Fanuc TP program (LS listing): CODE5.ls

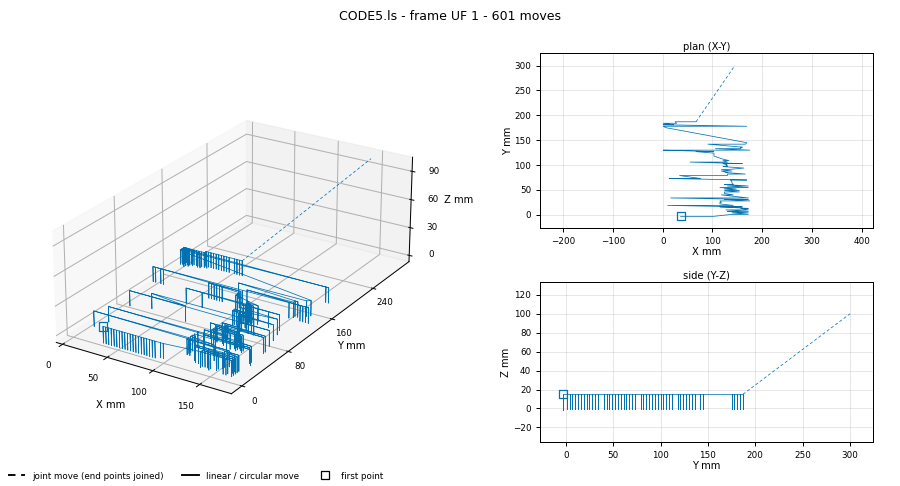
[picture p0: tool path of CODE5.ls in frame UF 1, 601 of 601 moves have a stored position in this frame; points joined in program order, loops and branches not executed]
/PROG CODE5
/ATTR
OWNER		= NOC_FANU;
COMMENT		= "NOC_FANUC";
PROG_SIZE	= 328;
CREATE		= DATE 97-07-08  TIME 03:05:20;
MODIFIED	= DATE 17-07-08  TIME 03:05:26;
FILE_NAME	= ;
VERSION		= 0;
LINE_COUNT	= 10;
MEMORY_SIZE	= 692;
PROTECT		= READ_WRITE;
TCD:  STACK_SIZE	= 0,
      TASK_PRIORITY	= 0,
      TIME_SLICE	= 0,
      BUSY_LAMP_OFF	= 0,
      ABORT_REQUEST	= 0,
      PAUSE_REQUEST	= 0;
DEFAULT_GROUP	= 1,*,*,*,*;
CONTROL_CODE	= 00000000 00000000;
/APPL
/MN
1:UFRAME_NUM=1 ;
2:UTOOL_NUM=5;
3:J P[265] 10% CNT100;
4:L P[266] 250mm/sec FINE;
5:L P[267] 250mm/sec CNT100;
6:L P[268] 250mm/sec CNT100;
7:L P[269] 250mm/sec FINE;
8:L P[270] 250mm/sec CNT100;
9:L P[271] 250mm/sec CNT100;
10:L P[272] 250mm/sec FINE;
11:L P[273] 250mm/sec CNT100;
12:L P[274] 250mm/sec CNT100;
13:L P[275] 250mm/sec FINE;
14:L P[276] 250mm/sec CNT100;
15:L P[277] 250mm/sec CNT100;
16:L P[278] 250mm/sec FINE;
17:L P[279] 250mm/sec CNT100;
18:L P[280] 250mm/sec CNT100;
19:L P[281] 250mm/sec FINE;
20:L P[282] 250mm/sec CNT100;
21:L P[283] 250mm/sec CNT100;
22:L P[284] 250mm/sec FINE;
23:L P[285] 250mm/sec CNT100;
24:L P[286] 250mm/sec CNT100;
25:L P[287] 250mm/sec FINE;
26:L P[288] 250mm/sec CNT100;
27:L P[289] 250mm/sec CNT100;
28:L P[290] 250mm/sec FINE;
29:L P[291] 250mm/sec CNT100;
30:L P[292] 250mm/sec CNT100;
31:L P[293] 250mm/sec FINE;
32:L P[294] 250mm/sec CNT100;
33:L P[295] 250mm/sec CNT100;
34:L P[296] 250mm/sec FINE;
35:L P[297] 250mm/sec CNT100;
36:L P[298] 250mm/sec CNT100;
37:L P[299] 250mm/sec FINE;
38:L P[300] 250mm/sec CNT100;
39:L P[301] 250mm/sec CNT100;
40:L P[302] 250mm/sec FINE;
41:L P[303] 250mm/sec CNT100;
42:L P[304] 250mm/sec CNT100;
43:L P[305] 250mm/sec FINE;
44:L P[306] 250mm/sec CNT100;
45:L P[307] 250mm/sec CNT100;
46:L P[308] 250mm/sec FINE;
47:L P[309] 250mm/sec CNT100;
48:L P[310] 250mm/sec CNT100;
49:L P[311] 250mm/sec FINE;
50:L P[312] 250mm/sec CNT100;
51:L P[313] 250mm/sec CNT100;
52:L P[314] 250mm/sec FINE;
53:L P[315] 250mm/sec CNT100;
54:L P[316] 250mm/sec CNT100;
55:L P[317] 250mm/sec FINE;
56:L P[318] 250mm/sec CNT100;
57:L P[319] 250mm/sec CNT100;
58:L P[320] 250mm/sec FINE;
59:L P[321] 250mm/sec CNT100;
60:L P[322] 250mm/sec CNT100;
61:L P[323] 250mm/sec FINE;
62:L P[324] 250mm/sec CNT100;
63:L P[325] 250mm/sec CNT100;
64:L P[326] 250mm/sec FINE;
65:L P[327] 250mm/sec CNT100;
66:L P[328] 250mm/sec CNT100;
67:L P[329] 250mm/sec FINE;
68:L P[330] 250mm/sec CNT100;
69:L P[535] 250mm/sec CNT100;
70:L P[536] 250mm/sec FINE;
71:L P[537] 250mm/sec CNT100;
72:L P[538] 250mm/sec CNT100;
73:L P[539] 250mm/sec FINE;
74:L P[540] 250mm/sec CNT100;
75:L P[541] 250mm/sec CNT100;
76:L P[542] 250mm/sec FINE;
77:L P[543] 250mm/sec CNT100;
78:L P[544] 250mm/sec CNT100;
79:L P[545] 250mm/sec FINE;
80:L P[546] 250mm/sec CNT100;
81:L P[550] 250mm/sec CNT100;
82:L P[551] 250mm/sec FINE;
83:L P[552] 250mm/sec CNT100;
84:L P[697] 250mm/sec CNT100;
85:L P[698] 250mm/sec FINE;
86:L P[699] 250mm/sec CNT100;
87:L P[700] 250mm/sec CNT100;
88:L P[701] 250mm/sec FINE;
89:L P[702] 250mm/sec CNT100;
90:L P[703] 250mm/sec CNT100;
91:L P[704] 250mm/sec FINE;
92:L P[705] 250mm/sec CNT100;
93:L P[706] 250mm/sec CNT100;
94:L P[707] 250mm/sec FINE;
95:L P[708] 250mm/sec CNT100;
96:L P[712] 250mm/sec CNT100;
97:L P[713] 250mm/sec FINE;
98:L P[714] 250mm/sec CNT100;
99:L P[715] 250mm/sec CNT100;
100:L P[716] 250mm/sec FINE;
101:L P[717] 250mm/sec CNT100;
102:L P[718] 250mm/sec CNT100;
103:L P[719] 250mm/sec FINE;
104:L P[720] 250mm/sec CNT100;
105:L P[856] 250mm/sec CNT100;
106:L P[857] 250mm/sec FINE;
107:L P[858] 250mm/sec CNT100;
108:L P[859] 250mm/sec CNT100;
109:L P[860] 250mm/sec FINE;
110:L P[861] 250mm/sec CNT100;
111:L P[868] 250mm/sec CNT100;
112:L P[869] 250mm/sec FINE;
113:L P[870] 250mm/sec CNT100;
114:L P[874] 250mm/sec CNT100;
115:L P[875] 250mm/sec FINE;
116:L P[876] 250mm/sec CNT100;
117:L P[877] 250mm/sec CNT100;
118:L P[878] 250mm/sec FINE;
119:L P[879] 250mm/sec CNT100;
120:L P[1012] 250mm/sec CNT100;
121:L P[1013] 250mm/sec FINE;
122:L P[1014] 250mm/sec CNT100;
123:L P[1027] 250mm/sec CNT100;
124:L P[1028] 250mm/sec FINE;
125:L P[1029] 250mm/sec CNT100;
126:L P[1033] 250mm/sec CNT100;
127:L P[1034] 250mm/sec FINE;
128:L P[1035] 250mm/sec CNT100;
129:L P[1036] 250mm/sec CNT100;
130:L P[1037] 250mm/sec FINE;
131:L P[1038] 250mm/sec CNT100;
132:L P[1039] 250mm/sec CNT100;
133:L P[1040] 250mm/sec FINE;
134:L P[1041] 250mm/sec CNT100;
135:L P[1192] 250mm/sec CNT100;
136:L P[1193] 250mm/sec FINE;
137:L P[1194] 250mm/sec CNT100;
138:L P[1195] 250mm/sec CNT100;
139:L P[1196] 250mm/sec FINE;
140:L P[1197] 250mm/sec CNT100;
141:L P[1198] 250mm/sec CNT100;
142:L P[1199] 250mm/sec FINE;
143:L P[1200] 250mm/sec CNT100;
144:L P[1318] 250mm/sec CNT100;
145:L P[1319] 250mm/sec FINE;
146:L P[1320] 250mm/sec CNT100;
147:L P[1321] 250mm/sec CNT100;
148:L P[1322] 250mm/sec FINE;
149:L P[1323] 250mm/sec CNT100;
150:L P[1348] 250mm/sec CNT100;
151:L P[1349] 250mm/sec FINE;
152:L P[1350] 250mm/sec CNT100;
153:L P[1369] 250mm/sec CNT100;
154:L P[1370] 250mm/sec FINE;
155:L P[1371] 250mm/sec CNT100;
156:L P[1474] 250mm/sec CNT100;
157:L P[1475] 250mm/sec FINE;
158:L P[1476] 250mm/sec CNT100;
159:L P[1501] 250mm/sec CNT100;
160:L P[1502] 250mm/sec FINE;
161:L P[1503] 250mm/sec CNT100;
162:L P[1624] 250mm/sec CNT100;
163:L P[1625] 250mm/sec FINE;
164:L P[1626] 250mm/sec CNT100;
165:L P[1771] 250mm/sec CNT100;
166:L P[1772] 250mm/sec FINE;
167:L P[1773] 250mm/sec CNT100;
168:L P[1774] 250mm/sec CNT100;
169:L P[1775] 250mm/sec FINE;
170:L P[1776] 250mm/sec CNT100;
171:L P[1915] 250mm/sec CNT100;
172:L P[1916] 250mm/sec FINE;
173:L P[1917] 250mm/sec CNT100;
174:L P[1945] 250mm/sec CNT100;
175:L P[1946] 250mm/sec FINE;
176:L P[1947] 250mm/sec CNT100;
177:L P[2071] 250mm/sec CNT100;
178:L P[2072] 250mm/sec FINE;
179:L P[2073] 250mm/sec CNT100;
180:L P[2083] 250mm/sec CNT100;
181:L P[2084] 250mm/sec FINE;
182:L P[2085] 250mm/sec CNT100;
183:L P[2092] 250mm/sec CNT100;
184:L P[2093] 250mm/sec FINE;
185:L P[2094] 250mm/sec CNT100;
186:L P[2116] 250mm/sec CNT100;
187:L P[2117] 250mm/sec FINE;
188:L P[2118] 250mm/sec CNT100;
189:L P[2215] 250mm/sec CNT100;
190:L P[2216] 250mm/sec FINE;
191:L P[2217] 250mm/sec CNT100;
192:L P[2221] 250mm/sec CNT100;
193:L P[2222] 250mm/sec FINE;
194:L P[2223] 250mm/sec CNT100;
195:L P[2248] 250mm/sec CNT100;
196:L P[2249] 250mm/sec FINE;
197:L P[2250] 250mm/sec CNT100;
198:L P[2509] 250mm/sec CNT100;
199:L P[2510] 250mm/sec FINE;
200:L P[2511] 250mm/sec CNT100;
201:L P[2530] 250mm/sec CNT100;
202:L P[2531] 250mm/sec FINE;
203:L P[2532] 250mm/sec CNT100;
204:L P[2650] 250mm/sec CNT100;
205:L P[2651] 250mm/sec FINE;
206:L P[2652] 250mm/sec CNT100;
207:L P[2791] 250mm/sec CNT100;
208:L P[2792] 250mm/sec FINE;
209:L P[2793] 250mm/sec CNT100;
210:L P[2809] 250mm/sec CNT100;
211:L P[2810] 250mm/sec FINE;
212:L P[2811] 250mm/sec CNT100;
213:L P[2815] 250mm/sec CNT100;
214:L P[2816] 250mm/sec FINE;
215:L P[2817] 250mm/sec CNT100;
216:L P[2818] 250mm/sec CNT100;
217:L P[2819] 250mm/sec FINE;
218:L P[2820] 250mm/sec CNT100;
219:L P[2947] 250mm/sec CNT100;
220:L P[2948] 250mm/sec FINE;
221:L P[2949] 250mm/sec CNT100;
222:L P[2956] 250mm/sec CNT100;
223:L P[2957] 250mm/sec FINE;
224:L P[2958] 250mm/sec CNT100;
225:L P[2968] 250mm/sec CNT100;
226:L P[2969] 250mm/sec FINE;
227:L P[2970] 250mm/sec CNT100;
228:L P[2971] 250mm/sec CNT100;
229:L P[2972] 250mm/sec FINE;
230:L P[2973] 250mm/sec CNT100;
231:L P[2974] 250mm/sec CNT100;
232:L P[2975] 250mm/sec FINE;
233:L P[2976] 250mm/sec CNT100;
234:L P[2977] 250mm/sec CNT100;
235:L P[2978] 250mm/sec FINE;
236:L P[2979] 250mm/sec CNT100;
237:L P[3103] 250mm/sec CNT100;
238:L P[3104] 250mm/sec FINE;
239:L P[3105] 250mm/sec CNT100;
240:L P[3109] 250mm/sec CNT100;
241:L P[3110] 250mm/sec FINE;
242:L P[3111] 250mm/sec CNT100;
243:L P[3124] 250mm/sec CNT100;
244:L P[3125] 250mm/sec FINE;
245:L P[3126] 250mm/sec CNT100;
246:L P[3127] 250mm/sec CNT100;
247:L P[3128] 250mm/sec FINE;
248:L P[3129] 250mm/sec CNT100;
249:L P[3250] 250mm/sec CNT100;
250:L P[3251] 250mm/sec FINE;
251:L P[3252] 250mm/sec CNT100;
252:L P[3253] 250mm/sec CNT100;
253:L P[3254] 250mm/sec FINE;
254:L P[3255] 250mm/sec CNT100;
255:L P[3274] 250mm/sec CNT100;
256:L P[3275] 250mm/sec FINE;
257:L P[3276] 250mm/sec CNT100;
258:L P[3403] 250mm/sec CNT100;
259:L P[3404] 250mm/sec FINE;
260:L P[3405] 250mm/sec CNT100;
261:L P[3418] 250mm/sec CNT100;
262:L P[3419] 250mm/sec FINE;
263:L P[3420] 250mm/sec CNT100;
264:L P[3541] 250mm/sec CNT100;
265:L P[3542] 250mm/sec FINE;
266:L P[3543] 250mm/sec CNT100;
267:L P[3544] 250mm/sec CNT100;
268:L P[3545] 250mm/sec FINE;
269:L P[3546] 250mm/sec CNT100;
270:L P[3547] 250mm/sec CNT100;
271:L P[3548] 250mm/sec FINE;
272:L P[3549] 250mm/sec CNT100;
273:L P[3556] 250mm/sec CNT100;
274:L P[3557] 250mm/sec FINE;
275:L P[3558] 250mm/sec CNT100;
276:L P[3700] 250mm/sec CNT100;
277:L P[3701] 250mm/sec FINE;
278:L P[3702] 250mm/sec CNT100;
279:L P[3838] 250mm/sec CNT100;
280:L P[3839] 250mm/sec FINE;
281:L P[3840] 250mm/sec CNT100;
282:L P[3973] 250mm/sec CNT100;
283:L P[3974] 250mm/sec FINE;
284:L P[3975] 250mm/sec CNT100;
285:L P[3985] 250mm/sec CNT100;
286:L P[3986] 250mm/sec FINE;
287:L P[3987] 250mm/sec CNT100;
288:L P[4009] 250mm/sec CNT100;
289:L P[4010] 250mm/sec FINE;
290:L P[4011] 250mm/sec CNT100;
291:L P[4069] 250mm/sec CNT100;
292:L P[4070] 250mm/sec FINE;
293:L P[4071] 250mm/sec CNT100;
294:L P[4291] 250mm/sec CNT100;
295:L P[4292] 250mm/sec FINE;
296:L P[4293] 250mm/sec CNT100;
297:L P[4369] 250mm/sec CNT100;
298:L P[4370] 250mm/sec FINE;
299:L P[4371] 250mm/sec CNT100;
300:L P[4510] 250mm/sec CNT100;
301:L P[4511] 250mm/sec FINE;
302:L P[4512] 250mm/sec CNT100;
303:L P[4519] 250mm/sec CNT100;
304:L P[4520] 250mm/sec FINE;
305:L P[4521] 250mm/sec CNT100;
306:L P[4525] 250mm/sec CNT100;
307:L P[4526] 250mm/sec FINE;
308:L P[4527] 250mm/sec CNT100;
309:L P[4528] 250mm/sec CNT100;
310:L P[4529] 250mm/sec FINE;
311:L P[4530] 250mm/sec CNT100;
312:L P[4657] 250mm/sec CNT100;
313:L P[4658] 250mm/sec FINE;
314:L P[4659] 250mm/sec CNT100;
315:L P[4660] 250mm/sec CNT100;
316:L P[4661] 250mm/sec FINE;
317:L P[4662] 250mm/sec CNT100;
318:L P[4807] 250mm/sec CNT100;
319:L P[4808] 250mm/sec FINE;
320:L P[4809] 250mm/sec CNT100;
321:L P[4813] 250mm/sec CNT100;
322:L P[4814] 250mm/sec FINE;
323:L P[4815] 250mm/sec CNT100;
324:L P[4819] 250mm/sec CNT100;
325:L P[4820] 250mm/sec FINE;
326:L P[4821] 250mm/sec CNT100;
327:L P[4948] 250mm/sec CNT100;
328:L P[4949] 250mm/sec FINE;
329:L P[4950] 250mm/sec CNT100;
330:L P[4951] 250mm/sec CNT100;
331:L P[4952] 250mm/sec FINE;
332:L P[4953] 250mm/sec CNT100;
333:L P[4954] 250mm/sec CNT100;
334:L P[4955] 250mm/sec FINE;
335:L P[4956] 250mm/sec CNT100;
336:L P[4957] 250mm/sec CNT100;
337:L P[4958] 250mm/sec FINE;
338:L P[4959] 250mm/sec CNT100;
339:L P[5110] 250mm/sec CNT100;
340:L P[5111] 250mm/sec FINE;
341:L P[5112] 250mm/sec CNT100;
342:L P[5248] 250mm/sec CNT100;
343:L P[5249] 250mm/sec FINE;
344:L P[5250] 250mm/sec CNT100;
345:L P[5251] 250mm/sec CNT100;
346:L P[5252] 250mm/sec FINE;
347:L P[5253] 250mm/sec CNT100;
348:L P[5257] 250mm/sec CNT100;
349:L P[5258] 250mm/sec FINE;
350:L P[5259] 250mm/sec CNT100;
351:L P[5422] 250mm/sec CNT100;
352:L P[5423] 250mm/sec FINE;
353:L P[5424] 250mm/sec CNT100;
354:L P[5425] 250mm/sec CNT100;
355:L P[5426] 250mm/sec FINE;
356:L P[5427] 250mm/sec CNT100;
357:L P[5584] 250mm/sec CNT100;
358:L P[5585] 250mm/sec FINE;
359:L P[5586] 250mm/sec CNT100;
360:L P[5587] 250mm/sec CNT100;
361:L P[5588] 250mm/sec FINE;
362:L P[5589] 250mm/sec CNT100;
363:L P[5590] 250mm/sec CNT100;
364:L P[5591] 250mm/sec FINE;
365:L P[5592] 250mm/sec CNT100;
366:L P[5593] 250mm/sec CNT100;
367:L P[5594] 250mm/sec FINE;
368:L P[5595] 250mm/sec CNT100;
369:L P[5599] 250mm/sec CNT100;
370:L P[5600] 250mm/sec FINE;
371:L P[5601] 250mm/sec CNT100;
372:L P[5611] 250mm/sec CNT100;
373:L P[5612] 250mm/sec FINE;
374:L P[5613] 250mm/sec CNT100;
375:L P[5614] 250mm/sec CNT100;
376:L P[5615] 250mm/sec FINE;
377:L P[5616] 250mm/sec CNT100;
378:L P[5689] 250mm/sec CNT100;
379:L P[5690] 250mm/sec FINE;
380:L P[5691] 250mm/sec CNT100;
381:L P[5692] 250mm/sec CNT100;
382:L P[5693] 250mm/sec FINE;
383:L P[5694] 250mm/sec CNT100;
384:L P[5713] 250mm/sec CNT100;
385:L P[5714] 250mm/sec FINE;
386:L P[5715] 250mm/sec CNT100;
387:L P[5716] 250mm/sec CNT100;
388:L P[5717] 250mm/sec FINE;
389:L P[5718] 250mm/sec CNT100;
390:L P[5719] 250mm/sec CNT100;
391:L P[5720] 250mm/sec FINE;
392:L P[5721] 250mm/sec CNT100;
393:L P[5722] 250mm/sec CNT100;
394:L P[5723] 250mm/sec FINE;
395:L P[5724] 250mm/sec CNT100;
396:L P[5827] 250mm/sec CNT100;
397:L P[5828] 250mm/sec FINE;
398:L P[5829] 250mm/sec CNT100;
399:L P[5830] 250mm/sec CNT100;
400:L P[5831] 250mm/sec FINE;
401:L P[5832] 250mm/sec CNT100;
402:L P[5839] 250mm/sec CNT100;
403:L P[5840] 250mm/sec FINE;
404:L P[5841] 250mm/sec CNT100;
405:L P[5926] 250mm/sec CNT100;
406:L P[5927] 250mm/sec FINE;
407:L P[5928] 250mm/sec CNT100;
408:L P[6103] 250mm/sec CNT100;
409:L P[6104] 250mm/sec FINE;
410:L P[6105] 250mm/sec CNT100;
411:L P[6208] 250mm/sec CNT100;
412:L P[6209] 250mm/sec FINE;
413:L P[6210] 250mm/sec CNT100;
414:L P[6322] 250mm/sec CNT100;
415:L P[6323] 250mm/sec FINE;
416:L P[6324] 250mm/sec CNT100;
417:L P[6430] 250mm/sec CNT100;
418:L P[6431] 250mm/sec FINE;
419:L P[6432] 250mm/sec CNT100;
420:L P[6433] 250mm/sec CNT100;
421:L P[6434] 250mm/sec FINE;
422:L P[6435] 250mm/sec CNT100;
423:L P[6436] 250mm/sec CNT100;
424:L P[6437] 250mm/sec FINE;
425:L P[6438] 250mm/sec CNT100;
426:L P[6439] 250mm/sec CNT100;
427:L P[6440] 250mm/sec FINE;
428:L P[6441] 250mm/sec CNT100;
429:L P[6442] 250mm/sec CNT100;
430:L P[6443] 250mm/sec FINE;
431:L P[6444] 250mm/sec CNT100;
432:L P[6445] 250mm/sec CNT100;
433:L P[6446] 250mm/sec FINE;
434:L P[6447] 250mm/sec CNT100;
435:L P[6448] 250mm/sec CNT100;
436:L P[6449] 250mm/sec FINE;
437:L P[6450] 250mm/sec CNT100;
438:L P[6490] 250mm/sec CNT100;
439:L P[6491] 250mm/sec FINE;
440:L P[6492] 250mm/sec CNT100;
441:L P[6493] 250mm/sec CNT100;
442:L P[6494] 250mm/sec FINE;
443:L P[6495] 250mm/sec CNT100;
444:L P[6499] 250mm/sec CNT100;
445:L P[6500] 250mm/sec FINE;
446:L P[6501] 250mm/sec CNT100;
447:L P[6502] 250mm/sec CNT100;
448:L P[6503] 250mm/sec FINE;
449:L P[6504] 250mm/sec CNT100;
450:L P[6553] 250mm/sec CNT100;
451:L P[6554] 250mm/sec FINE;
452:L P[6555] 250mm/sec CNT100;
453:L P[6598] 250mm/sec CNT100;
454:L P[6599] 250mm/sec FINE;
455:L P[6600] 250mm/sec CNT100;
456:L P[6610] 250mm/sec CNT100;
457:L P[6611] 250mm/sec FINE;
458:L P[6612] 250mm/sec CNT100;
459:L P[6613] 250mm/sec CNT100;
460:L P[6614] 250mm/sec FINE;
461:L P[6615] 250mm/sec CNT100;
462:L P[6616] 250mm/sec CNT100;
463:L P[6617] 250mm/sec FINE;
464:L P[6618] 250mm/sec CNT100;
465:L P[6619] 250mm/sec CNT100;
466:L P[6620] 250mm/sec FINE;
467:L P[6621] 250mm/sec CNT100;
468:L P[6676] 250mm/sec CNT100;
469:L P[6677] 250mm/sec FINE;
470:L P[6678] 250mm/sec CNT100;
471:L P[6727] 250mm/sec CNT100;
472:L P[6728] 250mm/sec FINE;
473:L P[6729] 250mm/sec CNT100;
474:L P[6826] 250mm/sec CNT100;
475:L P[6827] 250mm/sec FINE;
476:L P[6828] 250mm/sec CNT100;
477:L P[6829] 250mm/sec CNT100;
478:L P[6830] 250mm/sec FINE;
479:L P[6831] 250mm/sec CNT100;
480:L P[6985] 250mm/sec CNT100;
481:L P[6986] 250mm/sec FINE;
482:L P[6987] 250mm/sec CNT100;
483:L P[7048] 250mm/sec CNT100;
484:L P[7049] 250mm/sec FINE;
485:L P[7050] 250mm/sec CNT100;
486:L P[7150] 250mm/sec CNT100;
487:L P[7151] 250mm/sec FINE;
488:L P[7152] 250mm/sec CNT100;
489:L P[7996] 250mm/sec CNT100;
490:L P[7997] 250mm/sec FINE;
491:L P[7998] 250mm/sec CNT100;
492:L P[8056] 250mm/sec CNT100;
493:L P[8057] 250mm/sec FINE;
494:L P[8058] 250mm/sec CNT100;
495:L P[8059] 250mm/sec CNT100;
496:L P[8060] 250mm/sec FINE;
497:L P[8061] 250mm/sec CNT100;
498:L P[8062] 250mm/sec CNT100;
499:L P[8063] 250mm/sec FINE;
500:L P[8064] 250mm/sec CNT100;
501:L P[8065] 250mm/sec CNT100;
502:L P[8066] 250mm/sec FINE;
503:L P[8067] 250mm/sec CNT100;
504:L P[8119] 250mm/sec CNT100;
505:L P[8120] 250mm/sec FINE;
506:L P[8121] 250mm/sec CNT100;
507:L P[8122] 250mm/sec CNT100;
508:L P[8123] 250mm/sec FINE;
509:L P[8124] 250mm/sec CNT100;
510:L P[8134] 250mm/sec CNT100;
511:L P[8135] 250mm/sec FINE;
512:L P[8136] 250mm/sec CNT100;
513:L P[8137] 250mm/sec CNT100;
514:L P[8138] 250mm/sec FINE;
515:L P[8139] 250mm/sec CNT100;
516:L P[8140] 250mm/sec CNT100;
517:L P[8141] 250mm/sec FINE;
518:L P[8142] 250mm/sec CNT100;
519:L P[8143] 250mm/sec CNT100;
520:L P[8144] 250mm/sec FINE;
521:L P[8145] 250mm/sec CNT100;
522:L P[8146] 250mm/sec CNT100;
523:L P[8147] 250mm/sec FINE;
524:L P[8148] 250mm/sec CNT100;
525:L P[8152] 250mm/sec CNT100;
526:L P[8153] 250mm/sec FINE;
527:L P[8154] 250mm/sec CNT100;
528:L P[8155] 250mm/sec CNT100;
529:L P[8156] 250mm/sec FINE;
530:L P[8157] 250mm/sec CNT100;
531:L P[8230] 250mm/sec CNT100;
532:L P[8231] 250mm/sec FINE;
533:L P[8232] 250mm/sec CNT100;
534:L P[8233] 250mm/sec CNT100;
535:L P[8234] 250mm/sec FINE;
536:L P[8235] 250mm/sec CNT100;
537:L P[8236] 250mm/sec CNT100;
538:L P[8237] 250mm/sec FINE;
539:L P[8238] 250mm/sec CNT100;
540:L P[8239] 250mm/sec CNT100;
541:L P[8240] 250mm/sec FINE;
542:L P[8241] 250mm/sec CNT100;
543:L P[8242] 250mm/sec CNT100;
544:L P[8243] 250mm/sec FINE;
545:L P[8244] 250mm/sec CNT100;
546:L P[8245] 250mm/sec CNT100;
547:L P[8246] 250mm/sec FINE;
548:L P[8247] 250mm/sec CNT100;
549:L P[8248] 250mm/sec CNT100;
550:L P[8249] 250mm/sec FINE;
551:L P[8250] 250mm/sec CNT100;
552:L P[8251] 250mm/sec CNT100;
553:L P[8252] 250mm/sec FINE;
554:L P[8253] 250mm/sec CNT100;
555:L P[8254] 250mm/sec CNT100;
556:L P[8255] 250mm/sec FINE;
557:L P[8256] 250mm/sec CNT100;
558:L P[8257] 250mm/sec CNT100;
559:L P[8258] 250mm/sec FINE;
560:L P[8259] 250mm/sec CNT100;
561:L P[8356] 250mm/sec CNT100;
562:L P[8357] 250mm/sec FINE;
563:L P[8358] 250mm/sec CNT100;
564:L P[8359] 250mm/sec CNT100;
565:L P[8360] 250mm/sec FINE;
566:L P[8361] 250mm/sec CNT100;
567:L P[8362] 250mm/sec CNT100;
568:L P[8363] 250mm/sec FINE;
569:L P[8364] 250mm/sec CNT100;
570:L P[8365] 250mm/sec CNT100;
571:L P[8366] 250mm/sec FINE;
572:L P[8367] 250mm/sec CNT100;
573:L P[8368] 250mm/sec CNT100;
574:L P[8369] 250mm/sec FINE;
575:L P[8370] 250mm/sec CNT100;
576:L P[8371] 250mm/sec CNT100;
577:L P[8372] 250mm/sec FINE;
578:L P[8373] 250mm/sec CNT100;
579:L P[8374] 250mm/sec CNT100;
580:L P[8375] 250mm/sec FINE;
581:L P[8376] 250mm/sec CNT100;
582:L P[8377] 250mm/sec CNT100;
583:L P[8378] 250mm/sec FINE;
584:L P[8379] 250mm/sec CNT100;
585:L P[8380] 250mm/sec CNT100;
586:L P[8381] 250mm/sec FINE;
587:L P[8382] 250mm/sec CNT100;
588:L P[8383] 250mm/sec CNT100;
589:L P[8384] 250mm/sec FINE;
590:L P[8385] 250mm/sec CNT100;
591:L P[8386] 250mm/sec CNT100;
592:L P[8387] 250mm/sec FINE;
593:L P[8388] 250mm/sec CNT100;
594:L P[8389] 250mm/sec CNT100;
595:L P[8390] 250mm/sec FINE;
596:L P[8391] 250mm/sec CNT100;
597:L P[8392] 250mm/sec CNT100;
598:L P[8393] 250mm/sec FINE;
599:L P[8394] 250mm/sec CNT100;
600:L P[8395] 250mm/sec CNT100;
601:L P[8396] 250mm/sec FINE;
602:L P[8397] 250mm/sec CNT100;
603:J P[11569] 50% CNT100;
/POS
P[265]{
   GP1:
	UF : 1, UT : 5,		CONFIG : 'N U T, 0, 0, 0',
	X =  36.000  mm,	Y =  -3.000  mm,	Z =   15.000 mm,
	W =-180.000 deg,	P =   0.000 deg,	R =    90.000 deg
};
P[266]{
   GP1:
	UF : 1, UT : 5,		CONFIG : 'N U T, 0, 0, 0',
	X =  36.000  mm,	Y =  -3.000  mm,	Z =   -2.000 mm,
	W =-180.000 deg,	P =   0.000 deg,	R =    90.000 deg
};
P[267]{
   GP1:
	UF : 1, UT : 5,		CONFIG : 'N U T, 0, 0, 0',
	X =  36.000  mm,	Y =  -3.000  mm,	Z =   15.000 mm,
	W =-180.000 deg,	P =   0.000 deg,	R =    90.000 deg
};
P[268]{
   GP1:
	UF : 1, UT : 5,		CONFIG : 'N U T, 0, 0, 0',
	X =  39.000  mm,	Y =  -3.000  mm,	Z =   15.000 mm,
	W =-180.000 deg,	P =   0.000 deg,	R =    90.000 deg
};
P[269]{
   GP1:
	UF : 1, UT : 5,		CONFIG : 'N U T, 0, 0, 0',
	X =  39.000  mm,	Y =  -3.000  mm,	Z =   -2.000 mm,
	W =-180.000 deg,	P =   0.000 deg,	R =    90.000 deg
};
P[270]{
   GP1:
	UF : 1, UT : 5,		CONFIG : 'N U T, 0, 0, 0',
	X =  39.000  mm,	Y =  -3.000  mm,	Z =   15.000 mm,
	W =-180.000 deg,	P =   0.000 deg,	R =    90.000 deg
};
P[271]{
   GP1:
	UF : 1, UT : 5,		CONFIG : 'N U T, 0, 0, 0',
	X =  42.000  mm,	Y =  -3.000  mm,	Z =   15.000 mm,
	W =-180.000 deg,	P =   0.000 deg,	R =    90.000 deg
};
P[272]{
   GP1:
	UF : 1, UT : 5,		CONFIG : 'N U T, 0, 0, 0',
	X =  42.000  mm,	Y =  -3.000  mm,	Z =   -2.000 mm,
	W =-180.000 deg,	P =   0.000 deg,	R =    90.000 deg
};
P[273]{
   GP1:
	UF : 1, UT : 5,		CONFIG : 'N U T, 0, 0, 0',
	X =  42.000  mm,	Y =  -3.000  mm,	Z =   15.000 mm,
	W =-180.000 deg,	P =   0.000 deg,	R =    90.000 deg
};
P[274]{
   GP1:
	UF : 1, UT : 5,		CONFIG : 'N U T, 0, 0, 0',
	X =  45.000  mm,	Y =  -3.000  mm,	Z =   15.000 mm,
	W =-180.000 deg,	P =   0.000 deg,	R =    90.000 deg
};
P[275]{
   GP1:
	UF : 1, UT : 5,		CONFIG : 'N U T, 0, 0, 0',
	X =  45.000  mm,	Y =  -3.000  mm,	Z =   -2.000 mm,
	W =-180.000 deg,	P =   0.000 deg,	R =    90.000 deg
};
P[276]{
   GP1:
	UF : 1, UT : 5,		CONFIG : 'N U T, 0, 0, 0',
	X =  45.000  mm,	Y =  -3.000  mm,	Z =   15.000 mm,
	W =-180.000 deg,	P =   0.000 deg,	R =    90.000 deg
};
P[277]{
   GP1:
	UF : 1, UT : 5,		CONFIG : 'N U T, 0, 0, 0',
	X =  48.000  mm,	Y =  -3.000  mm,	Z =   15.000 mm,
	W =-180.000 deg,	P =   0.000 deg,	R =    90.000 deg
};
P[278]{
   GP1:
	UF : 1, UT : 5,		CONFIG : 'N U T, 0, 0, 0',
	X =  48.000  mm,	Y =  -3.000  mm,	Z =   -2.000 mm,
	W =-180.000 deg,	P =   0.000 deg,	R =    90.000 deg
};
P[279]{
   GP1:
	UF : 1, UT : 5,		CONFIG : 'N U T, 0, 0, 0',
	X =  48.000  mm,	Y =  -3.000  mm,	Z =   15.000 mm,
	W =-180.000 deg,	P =   0.000 deg,	R =    90.000 deg
};
P[280]{
   GP1:
	UF : 1, UT : 5,		CONFIG : 'N U T, 0, 0, 0',
	X =  51.000  mm,	Y =  -3.000  mm,	Z =   15.000 mm,
	W =-180.000 deg,	P =   0.000 deg,	R =    90.000 deg
};
P[281]{
   GP1:
	UF : 1, UT : 5,		CONFIG : 'N U T, 0, 0, 0',
	X =  51.000  mm,	Y =  -3.000  mm,	Z =   -2.000 mm,
	W =-180.000 deg,	P =   0.000 deg,	R =    90.000 deg
};
P[282]{
   GP1:
	UF : 1, UT : 5,		CONFIG : 'N U T, 0, 0, 0',
	X =  51.000  mm,	Y =  -3.000  mm,	Z =   15.000 mm,
	W =-180.000 deg,	P =   0.000 deg,	R =    90.000 deg
};
P[283]{
   GP1:
	UF : 1, UT : 5,		CONFIG : 'N U T, 0, 0, 0',
	X =  54.000  mm,	Y =  -3.000  mm,	Z =   15.000 mm,
	W =-180.000 deg,	P =   0.000 deg,	R =    90.000 deg
};
P[284]{
   GP1:
	UF : 1, UT : 5,		CONFIG : 'N U T, 0, 0, 0',
	X =  54.000  mm,	Y =  -3.000  mm,	Z =   -2.000 mm,
	W =-180.000 deg,	P =   0.000 deg,	R =    90.000 deg
};
P[285]{
   GP1:
	UF : 1, UT : 5,		CONFIG : 'N U T, 0, 0, 0',
	X =  54.000  mm,	Y =  -3.000  mm,	Z =   15.000 mm,
	W =-180.000 deg,	P =   0.000 deg,	R =    90.000 deg
};
P[286]{
   GP1:
	UF : 1, UT : 5,		CONFIG : 'N U T, 0, 0, 0',
	X =  57.000  mm,	Y =  -3.000  mm,	Z =   15.000 mm,
	W =-180.000 deg,	P =   0.000 deg,	R =    90.000 deg
};
P[287]{
   GP1:
	UF : 1, UT : 5,		CONFIG : 'N U T, 0, 0, 0',
	X =  57.000  mm,	Y =  -3.000  mm,	Z =   -2.000 mm,
	W =-180.000 deg,	P =   0.000 deg,	R =    90.000 deg
};
P[288]{
   GP1:
	UF : 1, UT : 5,		CONFIG : 'N U T, 0, 0, 0',
	X =  57.000  mm,	Y =  -3.000  mm,	Z =   15.000 mm,
	W =-180.000 deg,	P =   0.000 deg,	R =    90.000 deg
};
P[289]{
   GP1:
	UF : 1, UT : 5,		CONFIG : 'N U T, 0, 0, 0',
	X =  60.000  mm,	Y =  -3.000  mm,	Z =   15.000 mm,
	W =-180.000 deg,	P =   0.000 deg,	R =    90.000 deg
};
P[290]{
   GP1:
	UF : 1, UT : 5,		CONFIG : 'N U T, 0, 0, 0',
	X =  60.000  mm,	Y =  -3.000  mm,	Z =   -2.000 mm,
	W =-180.000 deg,	P =   0.000 deg,	R =    90.000 deg
};
P[291]{
   GP1:
	UF : 1, UT : 5,		CONFIG : 'N U T, 0, 0, 0',
	X =  60.000  mm,	Y =  -3.000  mm,	Z =   15.000 mm,
	W =-180.000 deg,	P =   0.000 deg,	R =    90.000 deg
};
P[292]{
   GP1:
	UF : 1, UT : 5,		CONFIG : 'N U T, 0, 0, 0',
	X =  63.000  mm,	Y =  -3.000  mm,	Z =   15.000 mm,
	W =-180.000 deg,	P =   0.000 deg,	R =    90.000 deg
};
P[293]{
   GP1:
	UF : 1, UT : 5,		CONFIG : 'N U T, 0, 0, 0',
	X =  63.000  mm,	Y =  -3.000  mm,	Z =   -2.000 mm,
	W =-180.000 deg,	P =   0.000 deg,	R =    90.000 deg
};
P[294]{
   GP1:
	UF : 1, UT : 5,		CONFIG : 'N U T, 0, 0, 0',
	X =  63.000  mm,	Y =  -3.000  mm,	Z =   15.000 mm,
	W =-180.000 deg,	P =   0.000 deg,	R =    90.000 deg
};
P[295]{
   GP1:
	UF : 1, UT : 5,		CONFIG : 'N U T, 0, 0, 0',
	X =  66.000  mm,	Y =  -3.000  mm,	Z =   15.000 mm,
	W =-180.000 deg,	P =   0.000 deg,	R =    90.000 deg
};
P[296]{
   GP1:
	UF : 1, UT : 5,		CONFIG : 'N U T, 0, 0, 0',
	X =  66.000  mm,	Y =  -3.000  mm,	Z =   -2.000 mm,
	W =-180.000 deg,	P =   0.000 deg,	R =    90.000 deg
};
P[297]{
   GP1:
	UF : 1, UT : 5,		CONFIG : 'N U T, 0, 0, 0',
	X =  66.000  mm,	Y =  -3.000  mm,	Z =   15.000 mm,
	W =-180.000 deg,	P =   0.000 deg,	R =    90.000 deg
};
P[298]{
   GP1:
	UF : 1, UT : 5,		CONFIG : 'N U T, 0, 0, 0',
	X =  69.000  mm,	Y =  -3.000  mm,	Z =   15.000 mm,
	W =-180.000 deg,	P =   0.000 deg,	R =    90.000 deg
};
P[299]{
   GP1:
	UF : 1, UT : 5,		CONFIG : 'N U T, 0, 0, 0',
	X =  69.000  mm,	Y =  -3.000  mm,	Z =   -2.000 mm,
	W =-180.000 deg,	P =   0.000 deg,	R =    90.000 deg
};
P[300]{
   GP1:
	UF : 1, UT : 5,		CONFIG : 'N U T, 0, 0, 0',
	X =  69.000  mm,	Y =  -3.000  mm,	Z =   15.000 mm,
	W =-180.000 deg,	P =   0.000 deg,	R =    90.000 deg
};
P[301]{
   GP1:
	UF : 1, UT : 5,		CONFIG : 'N U T, 0, 0, 0',
	X =  72.000  mm,	Y =  -3.000  mm,	Z =   15.000 mm,
	W =-180.000 deg,	P =   0.000 deg,	R =    90.000 deg
};
P[302]{
   GP1:
	UF : 1, UT : 5,		CONFIG : 'N U T, 0, 0, 0',
	X =  72.000  mm,	Y =  -3.000  mm,	Z =   -2.000 mm,
	W =-180.000 deg,	P =   0.000 deg,	R =    90.000 deg
};
P[303]{
   GP1:
	UF : 1, UT : 5,		CONFIG : 'N U T, 0, 0, 0',
	X =  72.000  mm,	Y =  -3.000  mm,	Z =   15.000 mm,
	W =-180.000 deg,	P =   0.000 deg,	R =    90.000 deg
};
P[304]{
   GP1:
	UF : 1, UT : 5,		CONFIG : 'N U T, 0, 0, 0',
	X =  75.000  mm,	Y =  -3.000  mm,	Z =   15.000 mm,
	W =-180.000 deg,	P =   0.000 deg,	R =    90.000 deg
};
P[305]{
   GP1:
	UF : 1, UT : 5,		CONFIG : 'N U T, 0, 0, 0',
	X =  75.000  mm,	Y =  -3.000  mm,	Z =   -2.000 mm,
	W =-180.000 deg,	P =   0.000 deg,	R =    90.000 deg
};
P[306]{
   GP1:
	UF : 1, UT : 5,		CONFIG : 'N U T, 0, 0, 0',
	X =  75.000  mm,	Y =  -3.000  mm,	Z =   15.000 mm,
	W =-180.000 deg,	P =   0.000 deg,	R =    90.000 deg
};
P[307]{
   GP1:
	UF : 1, UT : 5,		CONFIG : 'N U T, 0, 0, 0',
	X =  78.000  mm,	Y =  -3.000  mm,	Z =   15.000 mm,
	W =-180.000 deg,	P =   0.000 deg,	R =    90.000 deg
};
P[308]{
   GP1:
	UF : 1, UT : 5,		CONFIG : 'N U T, 0, 0, 0',
	X =  78.000  mm,	Y =  -3.000  mm,	Z =   -2.000 mm,
	W =-180.000 deg,	P =   0.000 deg,	R =    90.000 deg
};
P[309]{
   GP1:
	UF : 1, UT : 5,		CONFIG : 'N U T, 0, 0, 0',
	X =  78.000  mm,	Y =  -3.000  mm,	Z =   15.000 mm,
	W =-180.000 deg,	P =   0.000 deg,	R =    90.000 deg
};
P[310]{
   GP1:
	UF : 1, UT : 5,		CONFIG : 'N U T, 0, 0, 0',
	X =  81.000  mm,	Y =  -3.000  mm,	Z =   15.000 mm,
	W =-180.000 deg,	P =   0.000 deg,	R =    90.000 deg
};
P[311]{
   GP1:
	UF : 1, UT : 5,		CONFIG : 'N U T, 0, 0, 0',
	X =  81.000  mm,	Y =  -3.000  mm,	Z =   -2.000 mm,
	W =-180.000 deg,	P =   0.000 deg,	R =    90.000 deg
};
P[312]{
   GP1:
	UF : 1, UT : 5,		CONFIG : 'N U T, 0, 0, 0',
	X =  81.000  mm,	Y =  -3.000  mm,	Z =   15.000 mm,
	W =-180.000 deg,	P =   0.000 deg,	R =    90.000 deg
};
P[313]{
   GP1:
	UF : 1, UT : 5,		CONFIG : 'N U T, 0, 0, 0',
	X =  84.000  mm,	Y =  -3.000  mm,	Z =   15.000 mm,
	W =-180.000 deg,	P =   0.000 deg,	R =    90.000 deg
};
P[314]{
   GP1:
	UF : 1, UT : 5,		CONFIG : 'N U T, 0, 0, 0',
	X =  84.000  mm,	Y =  -3.000  mm,	Z =   -2.000 mm,
	W =-180.000 deg,	P =   0.000 deg,	R =    90.000 deg
};
P[315]{
   GP1:
	UF : 1, UT : 5,		CONFIG : 'N U T, 0, 0, 0',
	X =  84.000  mm,	Y =  -3.000  mm,	Z =   15.000 mm,
	W =-180.000 deg,	P =   0.000 deg,	R =    90.000 deg
};
P[316]{
   GP1:
	UF : 1, UT : 5,		CONFIG : 'N U T, 0, 0, 0',
	X =  87.000  mm,	Y =  -3.000  mm,	Z =   15.000 mm,
	W =-180.000 deg,	P =   0.000 deg,	R =    90.000 deg
};
P[317]{
   GP1:
	UF : 1, UT : 5,		CONFIG : 'N U T, 0, 0, 0',
	X =  87.000  mm,	Y =  -3.000  mm,	Z =   -2.000 mm,
	W =-180.000 deg,	P =   0.000 deg,	R =    90.000 deg
};
P[318]{
   GP1:
	UF : 1, UT : 5,		CONFIG : 'N U T, 0, 0, 0',
	X =  87.000  mm,	Y =  -3.000  mm,	Z =   15.000 mm,
	W =-180.000 deg,	P =   0.000 deg,	R =    90.000 deg
};
P[319]{
   GP1:
	UF : 1, UT : 5,		CONFIG : 'N U T, 0, 0, 0',
	X =  90.000  mm,	Y =  -3.000  mm,	Z =   15.000 mm,
	W =-180.000 deg,	P =   0.000 deg,	R =    90.000 deg
};
P[320]{
   GP1:
	UF : 1, UT : 5,		CONFIG : 'N U T, 0, 0, 0',
	X =  90.000  mm,	Y =  -3.000  mm,	Z =   -2.000 mm,
	W =-180.000 deg,	P =   0.000 deg,	R =    90.000 deg
};
P[321]{
   GP1:
	UF : 1, UT : 5,		CONFIG : 'N U T, 0, 0, 0',
	X =  90.000  mm,	Y =  -3.000  mm,	Z =   15.000 mm,
	W =-180.000 deg,	P =   0.000 deg,	R =    90.000 deg
};
P[322]{
   GP1:
	UF : 1, UT : 5,		CONFIG : 'N U T, 0, 0, 0',
	X =  93.000  mm,	Y =  -3.000  mm,	Z =   15.000 mm,
	W =-180.000 deg,	P =   0.000 deg,	R =    90.000 deg
};
P[323]{
   GP1:
	UF : 1, UT : 5,		CONFIG : 'N U T, 0, 0, 0',
	X =  93.000  mm,	Y =  -3.000  mm,	Z =   -2.000 mm,
	W =-180.000 deg,	P =   0.000 deg,	R =    90.000 deg
};
P[324]{
   GP1:
	UF : 1, UT : 5,		CONFIG : 'N U T, 0, 0, 0',
	X =  93.000  mm,	Y =  -3.000  mm,	Z =   15.000 mm,
	W =-180.000 deg,	P =   0.000 deg,	R =    90.000 deg
};
P[325]{
   GP1:
	UF : 1, UT : 5,		CONFIG : 'N U T, 0, 0, 0',
	X =  99.000  mm,	Y =  -3.000  mm,	Z =   15.000 mm,
	W =-180.000 deg,	P =   0.000 deg,	R =    90.000 deg
};
P[326]{
   GP1:
	UF : 1, UT : 5,		CONFIG : 'N U T, 0, 0, 0',
	X =  99.000  mm,	Y =  -3.000  mm,	Z =   0.000 mm,
	W =-180.000 deg,	P =   0.000 deg,	R =    90.000 deg
};
P[327]{
   GP1:
	UF : 1, UT : 5,		CONFIG : 'N U T, 0, 0, 0',
	X =  99.000  mm,	Y =  -3.000  mm,	Z =   15.000 mm,
	W =-180.000 deg,	P =   0.000 deg,	R =    90.000 deg
};
P[328]{
   GP1:
	UF : 1, UT : 5,		CONFIG : 'N U T, 0, 0, 0',
	X =  102.000  mm,	Y =  -3.000  mm,	Z =   15.000 mm,
	W =-180.000 deg,	P =   0.000 deg,	R =    90.000 deg
};
P[329]{
   GP1:
	UF : 1, UT : 5,		CONFIG : 'N U T, 0, 0, 0',
	X =  102.000  mm,	Y =  -3.000  mm,	Z =   0.000 mm,
	W =-180.000 deg,	P =   0.000 deg,	R =    90.000 deg
};
P[330]{
   GP1:
	UF : 1, UT : 5,		CONFIG : 'N U T, 0, 0, 0',
	X =  102.000  mm,	Y =  -3.000  mm,	Z =   15.000 mm,
	W =-180.000 deg,	P =   0.000 deg,	R =    90.000 deg
};
P[535]{
   GP1:
	UF : 1, UT : 5,		CONFIG : 'N U T, 0, 0, 0',
	X =  139.000  mm,	Y =  1.000  mm,	Z =   15.000 mm,
	W =-180.000 deg,	P =   0.000 deg,	R =    90.000 deg
};
P[536]{
   GP1:
	UF : 1, UT : 5,		CONFIG : 'N U T, 0, 0, 0',
	X =  139.000  mm,	Y =  1.000  mm,	Z =   -1.000 mm,
	W =-180.000 deg,	P =   0.000 deg,	R =    90.000 deg
};
P[537]{
   GP1:
	UF : 1, UT : 5,		CONFIG : 'N U T, 0, 0, 0',
	X =  139.000  mm,	Y =  1.000  mm,	Z =   15.000 mm,
	W =-180.000 deg,	P =   0.000 deg,	R =    90.000 deg
};
P[538]{
   GP1:
	UF : 1, UT : 5,		CONFIG : 'N U T, 0, 0, 0',
	X =  148.000  mm,	Y =  1.000  mm,	Z =   15.000 mm,
	W =-180.000 deg,	P =   0.000 deg,	R =    90.000 deg
};
P[539]{
   GP1:
	UF : 1, UT : 5,		CONFIG : 'N U T, 0, 0, 0',
	X =  148.000  mm,	Y =  1.000  mm,	Z =   -1.000 mm,
	W =-180.000 deg,	P =   0.000 deg,	R =    90.000 deg
};
P[540]{
   GP1:
	UF : 1, UT : 5,		CONFIG : 'N U T, 0, 0, 0',
	X =  148.000  mm,	Y =  1.000  mm,	Z =   15.000 mm,
	W =-180.000 deg,	P =   0.000 deg,	R =    90.000 deg
};
P[541]{
   GP1:
	UF : 1, UT : 5,		CONFIG : 'N U T, 0, 0, 0',
	X =  163.000  mm,	Y =  1.000  mm,	Z =   15.000 mm,
	W =-180.000 deg,	P =   0.000 deg,	R =    90.000 deg
};
P[542]{
   GP1:
	UF : 1, UT : 5,		CONFIG : 'N U T, 0, 0, 0',
	X =  163.000  mm,	Y =  1.000  mm,	Z =   -1.000 mm,
	W =-180.000 deg,	P =   0.000 deg,	R =    90.000 deg
};
P[543]{
   GP1:
	UF : 1, UT : 5,		CONFIG : 'N U T, 0, 0, 0',
	X =  163.000  mm,	Y =  1.000  mm,	Z =   15.000 mm,
	W =-180.000 deg,	P =   0.000 deg,	R =    90.000 deg
};
P[544]{
   GP1:
	UF : 1, UT : 5,		CONFIG : 'N U T, 0, 0, 0',
	X =  166.000  mm,	Y =  1.000  mm,	Z =   15.000 mm,
	W =-180.000 deg,	P =   0.000 deg,	R =    90.000 deg
};
P[545]{
   GP1:
	UF : 1, UT : 5,		CONFIG : 'N U T, 0, 0, 0',
	X =  166.000  mm,	Y =  1.000  mm,	Z =   -1.000 mm,
	W =-180.000 deg,	P =   0.000 deg,	R =    90.000 deg
};
P[546]{
   GP1:
	UF : 1, UT : 5,		CONFIG : 'N U T, 0, 0, 0',
	X =  166.000  mm,	Y =  1.000  mm,	Z =   15.000 mm,
	W =-180.000 deg,	P =   0.000 deg,	R =    90.000 deg
};
P[550]{
   GP1:
	UF : 1, UT : 5,		CONFIG : 'N U T, 0, 0, 0',
	X =  172.000  mm,	Y =  1.000  mm,	Z =   15.000 mm,
	W =-180.000 deg,	P =   0.000 deg,	R =    90.000 deg
};
P[551]{
   GP1:
	UF : 1, UT : 5,		CONFIG : 'N U T, 0, 0, 0',
	X =  172.000  mm,	Y =  1.000  mm,	Z =   -1.000 mm,
	W =-180.000 deg,	P =   0.000 deg,	R =    90.000 deg
};
P[552]{
   GP1:
	UF : 1, UT : 5,		CONFIG : 'N U T, 0, 0, 0',
	X =  172.000  mm,	Y =  1.000  mm,	Z =   15.000 mm,
	W =-180.000 deg,	P =   0.000 deg,	R =    90.000 deg
};
P[697]{
   GP1:
	UF : 1, UT : 5,		CONFIG : 'N U T, 0, 0, 0',
	X =  139.000  mm,	Y =  4.000  mm,	Z =   15.000 mm,
	W =-180.000 deg,	P =   0.000 deg,	R =    90.000 deg
};
P[698]{
   GP1:
	UF : 1, UT : 5,		CONFIG : 'N U T, 0, 0, 0',
	X =  139.000  mm,	Y =  4.000  mm,	Z =   -1.000 mm,
	W =-180.000 deg,	P =   0.000 deg,	R =    90.000 deg
};
P[699]{
   GP1:
	UF : 1, UT : 5,		CONFIG : 'N U T, 0, 0, 0',
	X =  139.000  mm,	Y =  4.000  mm,	Z =   15.000 mm,
	W =-180.000 deg,	P =   0.000 deg,	R =    90.000 deg
};
P[700]{
   GP1:
	UF : 1, UT : 5,		CONFIG : 'N U T, 0, 0, 0',
	X =  142.000  mm,	Y =  4.000  mm,	Z =   15.000 mm,
	W =-180.000 deg,	P =   0.000 deg,	R =    90.000 deg
};
P[701]{
   GP1:
	UF : 1, UT : 5,		CONFIG : 'N U T, 0, 0, 0',
	X =  142.000  mm,	Y =  4.000  mm,	Z =   -1.000 mm,
	W =-180.000 deg,	P =   0.000 deg,	R =    90.000 deg
};
P[702]{
   GP1:
	UF : 1, UT : 5,		CONFIG : 'N U T, 0, 0, 0',
	X =  142.000  mm,	Y =  4.000  mm,	Z =   15.000 mm,
	W =-180.000 deg,	P =   0.000 deg,	R =    90.000 deg
};
P[703]{
   GP1:
	UF : 1, UT : 5,		CONFIG : 'N U T, 0, 0, 0',
	X =  145.000  mm,	Y =  4.000  mm,	Z =   15.000 mm,
	W =-180.000 deg,	P =   0.000 deg,	R =    90.000 deg
};
P[704]{
   GP1:
	UF : 1, UT : 5,		CONFIG : 'N U T, 0, 0, 0',
	X =  145.000  mm,	Y =  4.000  mm,	Z =   -1.000 mm,
	W =-180.000 deg,	P =   0.000 deg,	R =    90.000 deg
};
P[705]{
   GP1:
	UF : 1, UT : 5,		CONFIG : 'N U T, 0, 0, 0',
	X =  145.000  mm,	Y =  4.000  mm,	Z =   15.000 mm,
	W =-180.000 deg,	P =   0.000 deg,	R =    90.000 deg
};
P[706]{
   GP1:
	UF : 1, UT : 5,		CONFIG : 'N U T, 0, 0, 0',
	X =  148.000  mm,	Y =  4.000  mm,	Z =   15.000 mm,
	W =-180.000 deg,	P =   0.000 deg,	R =    90.000 deg
};
P[707]{
   GP1:
	UF : 1, UT : 5,		CONFIG : 'N U T, 0, 0, 0',
	X =  148.000  mm,	Y =  4.000  mm,	Z =   -1.000 mm,
	W =-180.000 deg,	P =   0.000 deg,	R =    90.000 deg
};
P[708]{
   GP1:
	UF : 1, UT : 5,		CONFIG : 'N U T, 0, 0, 0',
	X =  148.000  mm,	Y =  4.000  mm,	Z =   15.000 mm,
	W =-180.000 deg,	P =   0.000 deg,	R =    90.000 deg
};
P[712]{
   GP1:
	UF : 1, UT : 5,		CONFIG : 'N U T, 0, 0, 0',
	X =  154.000  mm,	Y =  4.000  mm,	Z =   15.000 mm,
	W =-180.000 deg,	P =   0.000 deg,	R =    90.000 deg
};
P[713]{
   GP1:
	UF : 1, UT : 5,		CONFIG : 'N U T, 0, 0, 0',
	X =  154.000  mm,	Y =  4.000  mm,	Z =   -1.000 mm,
	W =-180.000 deg,	P =   0.000 deg,	R =    90.000 deg
};
P[714]{
   GP1:
	UF : 1, UT : 5,		CONFIG : 'N U T, 0, 0, 0',
	X =  154.000  mm,	Y =  4.000  mm,	Z =   15.000 mm,
	W =-180.000 deg,	P =   0.000 deg,	R =    90.000 deg
};
P[715]{
   GP1:
	UF : 1, UT : 5,		CONFIG : 'N U T, 0, 0, 0',
	X =  166.000  mm,	Y =  4.000  mm,	Z =   15.000 mm,
	W =-180.000 deg,	P =   0.000 deg,	R =    90.000 deg
};
P[716]{
   GP1:
	UF : 1, UT : 5,		CONFIG : 'N U T, 0, 0, 0',
	X =  166.000  mm,	Y =  4.000  mm,	Z =   -1.000 mm,
	W =-180.000 deg,	P =   0.000 deg,	R =    90.000 deg
};
P[717]{
   GP1:
	UF : 1, UT : 5,		CONFIG : 'N U T, 0, 0, 0',
	X =  166.000  mm,	Y =  4.000  mm,	Z =   15.000 mm,
	W =-180.000 deg,	P =   0.000 deg,	R =    90.000 deg
};
P[718]{
   GP1:
	UF : 1, UT : 5,		CONFIG : 'N U T, 0, 0, 0',
	X =  172.000  mm,	Y =  4.000  mm,	Z =   15.000 mm,
	W =-180.000 deg,	P =   0.000 deg,	R =    90.000 deg
};
P[719]{
   GP1:
	UF : 1, UT : 5,		CONFIG : 'N U T, 0, 0, 0',
	X =  172.000  mm,	Y =  4.000  mm,	Z =   -1.000 mm,
	W =-180.000 deg,	P =   0.000 deg,	R =    90.000 deg
};
P[720]{
   GP1:
	UF : 1, UT : 5,		CONFIG : 'N U T, 0, 0, 0',
	X =  172.000  mm,	Y =  4.000  mm,	Z =   15.000 mm,
	W =-180.000 deg,	P =   0.000 deg,	R =    90.000 deg
};
P[856]{
   GP1:
	UF : 1, UT : 5,		CONFIG : 'N U T, 0, 0, 0',
	X =  130.000  mm,	Y =  7.000  mm,	Z =   15.000 mm,
	W =-180.000 deg,	P =   0.000 deg,	R =    90.000 deg
};
P[857]{
   GP1:
	UF : 1, UT : 5,		CONFIG : 'N U T, 0, 0, 0',
	X =  130.000  mm,	Y =  7.000  mm,	Z =   -1.000 mm,
	W =-180.000 deg,	P =   0.000 deg,	R =    90.000 deg
};
P[858]{
   GP1:
	UF : 1, UT : 5,		CONFIG : 'N U T, 0, 0, 0',
	X =  130.000  mm,	Y =  7.000  mm,	Z =   15.000 mm,
	W =-180.000 deg,	P =   0.000 deg,	R =    90.000 deg
};
P[859]{
   GP1:
	UF : 1, UT : 5,		CONFIG : 'N U T, 0, 0, 0',
	X =  133.000  mm,	Y =  7.000  mm,	Z =   15.000 mm,
	W =-180.000 deg,	P =   0.000 deg,	R =    90.000 deg
};
P[860]{
   GP1:
	UF : 1, UT : 5,		CONFIG : 'N U T, 0, 0, 0',
	X =  133.000  mm,	Y =  7.000  mm,	Z =   -1.000 mm,
	W =-180.000 deg,	P =   0.000 deg,	R =    90.000 deg
};
P[861]{
   GP1:
	UF : 1, UT : 5,		CONFIG : 'N U T, 0, 0, 0',
	X =  133.000  mm,	Y =  7.000  mm,	Z =   15.000 mm,
	W =-180.000 deg,	P =   0.000 deg,	R =    90.000 deg
};
P[868]{
   GP1:
	UF : 1, UT : 5,		CONFIG : 'N U T, 0, 0, 0',
	X =  154.000  mm,	Y =  7.000  mm,	Z =   15.000 mm,
	W =-180.000 deg,	P =   0.000 deg,	R =    90.000 deg
};
P[869]{
   GP1:
	UF : 1, UT : 5,		CONFIG : 'N U T, 0, 0, 0',
	X =  154.000  mm,	Y =  7.000  mm,	Z =   -1.000 mm,
	W =-180.000 deg,	P =   0.000 deg,	R =    90.000 deg
};
P[870]{
   GP1:
	UF : 1, UT : 5,		CONFIG : 'N U T, 0, 0, 0',
	X =  154.000  mm,	Y =  7.000  mm,	Z =   15.000 mm,
	W =-180.000 deg,	P =   0.000 deg,	R =    90.000 deg
};
P[874]{
   GP1:
	UF : 1, UT : 5,		CONFIG : 'N U T, 0, 0, 0',
	X =  169.000  mm,	Y =  7.000  mm,	Z =   15.000 mm,
	W =-180.000 deg,	P =   0.000 deg,	R =    90.000 deg
};
P[875]{
   GP1:
	UF : 1, UT : 5,		CONFIG : 'N U T, 0, 0, 0',
	X =  169.000  mm,	Y =  7.000  mm,	Z =   -1.000 mm,
	W =-180.000 deg,	P =   0.000 deg,	R =    90.000 deg
};
P[876]{
   GP1:
	UF : 1, UT : 5,		CONFIG : 'N U T, 0, 0, 0',
	X =  169.000  mm,	Y =  7.000  mm,	Z =   15.000 mm,
	W =-180.000 deg,	P =   0.000 deg,	R =    90.000 deg
};
P[877]{
   GP1:
	UF : 1, UT : 5,		CONFIG : 'N U T, 0, 0, 0',
	X =  172.000  mm,	Y =  7.000  mm,	Z =   15.000 mm,
	W =-180.000 deg,	P =   0.000 deg,	R =    90.000 deg
};
P[878]{
   GP1:
	UF : 1, UT : 5,		CONFIG : 'N U T, 0, 0, 0',
	X =  172.000  mm,	Y =  7.000  mm,	Z =   -1.000 mm,
	W =-180.000 deg,	P =   0.000 deg,	R =    90.000 deg
};
P[879]{
   GP1:
	UF : 1, UT : 5,		CONFIG : 'N U T, 0, 0, 0',
	X =  172.000  mm,	Y =  7.000  mm,	Z =   15.000 mm,
	W =-180.000 deg,	P =   0.000 deg,	R =    90.000 deg
};
P[1012]{
   GP1:
	UF : 1, UT : 5,		CONFIG : 'N U T, 0, 0, 0',
	X =  127.000  mm,	Y =  10.000  mm,	Z =   15.000 mm,
	W =-180.000 deg,	P =   0.000 deg,	R =    90.000 deg
};
P[1013]{
   GP1:
	UF : 1, UT : 5,		CONFIG : 'N U T, 0, 0, 0',
	X =  127.000  mm,	Y =  10.000  mm,	Z =   -1.000 mm,
	W =-180.000 deg,	P =   0.000 deg,	R =    90.000 deg
};
P[1014]{
   GP1:
	UF : 1, UT : 5,		CONFIG : 'N U T, 0, 0, 0',
	X =  127.000  mm,	Y =  10.000  mm,	Z =   15.000 mm,
	W =-180.000 deg,	P =   0.000 deg,	R =    90.000 deg
};
P[1027]{
   GP1:
	UF : 1, UT : 5,		CONFIG : 'N U T, 0, 0, 0',
	X =  142.000  mm,	Y =  10.000  mm,	Z =   15.000 mm,
	W =-180.000 deg,	P =   0.000 deg,	R =    90.000 deg
};
P[1028]{
   GP1:
	UF : 1, UT : 5,		CONFIG : 'N U T, 0, 0, 0',
	X =  142.000  mm,	Y =  10.000  mm,	Z =   -1.000 mm,
	W =-180.000 deg,	P =   0.000 deg,	R =    90.000 deg
};
P[1029]{
   GP1:
	UF : 1, UT : 5,		CONFIG : 'N U T, 0, 0, 0',
	X =  142.000  mm,	Y =  10.000  mm,	Z =   15.000 mm,
	W =-180.000 deg,	P =   0.000 deg,	R =    90.000 deg
};
P[1033]{
   GP1:
	UF : 1, UT : 5,		CONFIG : 'N U T, 0, 0, 0',
	X =  157.000  mm,	Y =  10.000  mm,	Z =   15.000 mm,
	W =-180.000 deg,	P =   0.000 deg,	R =    90.000 deg
};
P[1034]{
   GP1:
	UF : 1, UT : 5,		CONFIG : 'N U T, 0, 0, 0',
	X =  157.000  mm,	Y =  10.000  mm,	Z =   -1.000 mm,
	W =-180.000 deg,	P =   0.000 deg,	R =    90.000 deg
};
P[1035]{
   GP1:
	UF : 1, UT : 5,		CONFIG : 'N U T, 0, 0, 0',
	X =  157.000  mm,	Y =  10.000  mm,	Z =   15.000 mm,
	W =-180.000 deg,	P =   0.000 deg,	R =    90.000 deg
};
P[1036]{
   GP1:
	UF : 1, UT : 5,		CONFIG : 'N U T, 0, 0, 0',
	X =  169.000  mm,	Y =  10.000  mm,	Z =   15.000 mm,
	W =-180.000 deg,	P =   0.000 deg,	R =    90.000 deg
};
P[1037]{
   GP1:
	UF : 1, UT : 5,		CONFIG : 'N U T, 0, 0, 0',
	X =  169.000  mm,	Y =  10.000  mm,	Z =   -1.000 mm,
	W =-180.000 deg,	P =   0.000 deg,	R =    90.000 deg
};
P[1038]{
   GP1:
	UF : 1, UT : 5,		CONFIG : 'N U T, 0, 0, 0',
	X =  169.000  mm,	Y =  10.000  mm,	Z =   15.000 mm,
	W =-180.000 deg,	P =   0.000 deg,	R =    90.000 deg
};
P[1039]{
   GP1:
	UF : 1, UT : 5,		CONFIG : 'N U T, 0, 0, 0',
	X =  172.000  mm,	Y =  10.000  mm,	Z =   15.000 mm,
	W =-180.000 deg,	P =   0.000 deg,	R =    90.000 deg
};
P[1040]{
   GP1:
	UF : 1, UT : 5,		CONFIG : 'N U T, 0, 0, 0',
	X =  172.000  mm,	Y =  10.000  mm,	Z =   -1.000 mm,
	W =-180.000 deg,	P =   0.000 deg,	R =    90.000 deg
};
P[1041]{
   GP1:
	UF : 1, UT : 5,		CONFIG : 'N U T, 0, 0, 0',
	X =  172.000  mm,	Y =  10.000  mm,	Z =   15.000 mm,
	W =-180.000 deg,	P =   0.000 deg,	R =    90.000 deg
};
P[1192]{
   GP1:
	UF : 1, UT : 5,		CONFIG : 'N U T, 0, 0, 0',
	X =  157.000  mm,	Y =  13.000  mm,	Z =   15.000 mm,
	W =-180.000 deg,	P =   0.000 deg,	R =    90.000 deg
};
P[1193]{
   GP1:
	UF : 1, UT : 5,		CONFIG : 'N U T, 0, 0, 0',
	X =  157.000  mm,	Y =  13.000  mm,	Z =   -1.000 mm,
	W =-180.000 deg,	P =   0.000 deg,	R =    90.000 deg
};
P[1194]{
   GP1:
	UF : 1, UT : 5,		CONFIG : 'N U T, 0, 0, 0',
	X =  157.000  mm,	Y =  13.000  mm,	Z =   15.000 mm,
	W =-180.000 deg,	P =   0.000 deg,	R =    90.000 deg
};
P[1195]{
   GP1:
	UF : 1, UT : 5,		CONFIG : 'N U T, 0, 0, 0',
	X =  160.000  mm,	Y =  13.000  mm,	Z =   15.000 mm,
	W =-180.000 deg,	P =   0.000 deg,	R =    90.000 deg
};
P[1196]{
   GP1:
	UF : 1, UT : 5,		CONFIG : 'N U T, 0, 0, 0',
	X =  160.000  mm,	Y =  13.000  mm,	Z =   -1.000 mm,
	W =-180.000 deg,	P =   0.000 deg,	R =    90.000 deg
};
P[1197]{
   GP1:
	UF : 1, UT : 5,		CONFIG : 'N U T, 0, 0, 0',
	X =  160.000  mm,	Y =  13.000  mm,	Z =   15.000 mm,
	W =-180.000 deg,	P =   0.000 deg,	R =    90.000 deg
};
P[1198]{
   GP1:
	UF : 1, UT : 5,		CONFIG : 'N U T, 0, 0, 0',
	X =  172.000  mm,	Y =  13.000  mm,	Z =   15.000 mm,
	W =-180.000 deg,	P =   0.000 deg,	R =    90.000 deg
};
P[1199]{
   GP1:
	UF : 1, UT : 5,		CONFIG : 'N U T, 0, 0, 0',
	X =  172.000  mm,	Y =  13.000  mm,	Z =   -1.000 mm,
	W =-180.000 deg,	P =   0.000 deg,	R =    90.000 deg
};
P[1200]{
   GP1:
	UF : 1, UT : 5,		CONFIG : 'N U T, 0, 0, 0',
	X =  172.000  mm,	Y =  13.000  mm,	Z =   15.000 mm,
	W =-180.000 deg,	P =   0.000 deg,	R =    90.000 deg
};
P[1318]{
   GP1:
	UF : 1, UT : 5,		CONFIG : 'N U T, 0, 0, 0',
	X =  115.000  mm,	Y =  16.000  mm,	Z =   15.000 mm,
	W =-180.000 deg,	P =   0.000 deg,	R =    90.000 deg
};
P[1319]{
   GP1:
	UF : 1, UT : 5,		CONFIG : 'N U T, 0, 0, 0',
	X =  115.000  mm,	Y =  16.000  mm,	Z =   -1.000 mm,
	W =-180.000 deg,	P =   0.000 deg,	R =    90.000 deg
};
P[1320]{
   GP1:
	UF : 1, UT : 5,		CONFIG : 'N U T, 0, 0, 0',
	X =  115.000  mm,	Y =  16.000  mm,	Z =   15.000 mm,
	W =-180.000 deg,	P =   0.000 deg,	R =    90.000 deg
};
P[1321]{
   GP1:
	UF : 1, UT : 5,		CONFIG : 'N U T, 0, 0, 0',
	X =  118.000  mm,	Y =  16.000  mm,	Z =   15.000 mm,
	W =-180.000 deg,	P =   0.000 deg,	R =    90.000 deg
};
P[1322]{
   GP1:
	UF : 1, UT : 5,		CONFIG : 'N U T, 0, 0, 0',
	X =  118.000  mm,	Y =  16.000  mm,	Z =   -1.000 mm,
	W =-180.000 deg,	P =   0.000 deg,	R =    90.000 deg
};
P[1323]{
   GP1:
	UF : 1, UT : 5,		CONFIG : 'N U T, 0, 0, 0',
	X =  118.000  mm,	Y =  16.000  mm,	Z =   15.000 mm,
	W =-180.000 deg,	P =   0.000 deg,	R =    90.000 deg
};
P[1348]{
   GP1:
	UF : 1, UT : 5,		CONFIG : 'N U T, 0, 0, 0',
	X =  160.000  mm,	Y =  16.000  mm,	Z =   15.000 mm,
	W =-180.000 deg,	P =   0.000 deg,	R =    90.000 deg
};
P[1349]{
   GP1:
	UF : 1, UT : 5,		CONFIG : 'N U T, 0, 0, 0',
	X =  160.000  mm,	Y =  16.000  mm,	Z =   -1.000 mm,
	W =-180.000 deg,	P =   0.000 deg,	R =    90.000 deg
};
P[1350]{
   GP1:
	UF : 1, UT : 5,		CONFIG : 'N U T, 0, 0, 0',
	X =  160.000  mm,	Y =  16.000  mm,	Z =   15.000 mm,
	W =-180.000 deg,	P =   0.000 deg,	R =    90.000 deg
};
P[1369]{
   GP1:
	UF : 1, UT : 5,		CONFIG : 'N U T, 0, 0, 0',
	X =  10.000  mm,	Y =  19.000  mm,	Z =   15.000 mm,
	W =-180.000 deg,	P =   0.000 deg,	R =    90.000 deg
};
P[1370]{
   GP1:
	UF : 1, UT : 5,		CONFIG : 'N U T, 0, 0, 0',
	X =  10.000  mm,	Y =  19.000  mm,	Z =   -1.000 mm,
	W =-180.000 deg,	P =   0.000 deg,	R =    90.000 deg
};
P[1371]{
   GP1:
	UF : 1, UT : 5,		CONFIG : 'N U T, 0, 0, 0',
	X =  10.000  mm,	Y =  19.000  mm,	Z =   15.000 mm,
	W =-180.000 deg,	P =   0.000 deg,	R =    90.000 deg
};
P[1474]{
   GP1:
	UF : 1, UT : 5,		CONFIG : 'N U T, 0, 0, 0',
	X =  115.000  mm,	Y =  19.000  mm,	Z =   15.000 mm,
	W =-180.000 deg,	P =   0.000 deg,	R =    90.000 deg
};
P[1475]{
   GP1:
	UF : 1, UT : 5,		CONFIG : 'N U T, 0, 0, 0',
	X =  115.000  mm,	Y =  19.000  mm,	Z =   -1.000 mm,
	W =-180.000 deg,	P =   0.000 deg,	R =    90.000 deg
};
P[1476]{
   GP1:
	UF : 1, UT : 5,		CONFIG : 'N U T, 0, 0, 0',
	X =  115.000  mm,	Y =  19.000  mm,	Z =   15.000 mm,
	W =-180.000 deg,	P =   0.000 deg,	R =    90.000 deg
};
P[1501]{
   GP1:
	UF : 1, UT : 5,		CONFIG : 'N U T, 0, 0, 0',
	X =  142.000  mm,	Y =  19.000  mm,	Z =   15.000 mm,
	W =-180.000 deg,	P =   0.000 deg,	R =    90.000 deg
};
P[1502]{
   GP1:
	UF : 1, UT : 5,		CONFIG : 'N U T, 0, 0, 0',
	X =  142.000  mm,	Y =  19.000  mm,	Z =   -1.000 mm,
	W =-180.000 deg,	P =   0.000 deg,	R =    90.000 deg
};
P[1503]{
   GP1:
	UF : 1, UT : 5,		CONFIG : 'N U T, 0, 0, 0',
	X =  142.000  mm,	Y =  19.000  mm,	Z =   15.000 mm,
	W =-180.000 deg,	P =   0.000 deg,	R =    90.000 deg
};
P[1624]{
   GP1:
	UF : 1, UT : 5,		CONFIG : 'N U T, 0, 0, 0',
	X =  115.000  mm,	Y =  22.000  mm,	Z =   15.000 mm,
	W =-180.000 deg,	P =   0.000 deg,	R =    90.000 deg
};
P[1625]{
   GP1:
	UF : 1, UT : 5,		CONFIG : 'N U T, 0, 0, 0',
	X =  115.000  mm,	Y =  22.000  mm,	Z =   -1.000 mm,
	W =-180.000 deg,	P =   0.000 deg,	R =    90.000 deg
};
P[1626]{
   GP1:
	UF : 1, UT : 5,		CONFIG : 'N U T, 0, 0, 0',
	X =  115.000  mm,	Y =  22.000  mm,	Z =   15.000 mm,
	W =-180.000 deg,	P =   0.000 deg,	R =    90.000 deg
};
P[1771]{
   GP1:
	UF : 1, UT : 5,		CONFIG : 'N U T, 0, 0, 0',
	X =  115.000  mm,	Y =  25.000  mm,	Z =   15.000 mm,
	W =-180.000 deg,	P =   0.000 deg,	R =    90.000 deg
};
P[1772]{
   GP1:
	UF : 1, UT : 5,		CONFIG : 'N U T, 0, 0, 0',
	X =  115.000  mm,	Y =  25.000  mm,	Z =   -1.000 mm,
	W =-180.000 deg,	P =   0.000 deg,	R =    90.000 deg
};
P[1773]{
   GP1:
	UF : 1, UT : 5,		CONFIG : 'N U T, 0, 0, 0',
	X =  115.000  mm,	Y =  25.000  mm,	Z =   15.000 mm,
	W =-180.000 deg,	P =   0.000 deg,	R =    90.000 deg
};
P[1774]{
   GP1:
	UF : 1, UT : 5,		CONFIG : 'N U T, 0, 0, 0',
	X =  118.000  mm,	Y =  25.000  mm,	Z =   15.000 mm,
	W =-180.000 deg,	P =   0.000 deg,	R =    90.000 deg
};
P[1775]{
   GP1:
	UF : 1, UT : 5,		CONFIG : 'N U T, 0, 0, 0',
	X =  118.000  mm,	Y =  25.000  mm,	Z =   -1.000 mm,
	W =-180.000 deg,	P =   0.000 deg,	R =    90.000 deg
};
P[1776]{
   GP1:
	UF : 1, UT : 5,		CONFIG : 'N U T, 0, 0, 0',
	X =  118.000  mm,	Y =  25.000  mm,	Z =   15.000 mm,
	W =-180.000 deg,	P =   0.000 deg,	R =    90.000 deg
};
P[1915]{
   GP1:
	UF : 1, UT : 5,		CONFIG : 'N U T, 0, 0, 0',
	X =  115.000  mm,	Y =  28.000  mm,	Z =   15.000 mm,
	W =-180.000 deg,	P =   0.000 deg,	R =    90.000 deg
};
P[1916]{
   GP1:
	UF : 1, UT : 5,		CONFIG : 'N U T, 0, 0, 0',
	X =  115.000  mm,	Y =  28.000  mm,	Z =   -1.000 mm,
	W =-180.000 deg,	P =   0.000 deg,	R =    90.000 deg
};
P[1917]{
   GP1:
	UF : 1, UT : 5,		CONFIG : 'N U T, 0, 0, 0',
	X =  115.000  mm,	Y =  28.000  mm,	Z =   15.000 mm,
	W =-180.000 deg,	P =   0.000 deg,	R =    90.000 deg
};
P[1945]{
   GP1:
	UF : 1, UT : 5,		CONFIG : 'N U T, 0, 0, 0',
	X =  175.000  mm,	Y =  28.000  mm,	Z =   15.000 mm,
	W =-180.000 deg,	P =   0.000 deg,	R =    90.000 deg
};
P[1946]{
   GP1:
	UF : 1, UT : 5,		CONFIG : 'N U T, 0, 0, 0',
	X =  175.000  mm,	Y =  28.000  mm,	Z =   -1.000 mm,
	W =-180.000 deg,	P =   0.000 deg,	R =    90.000 deg
};
P[1947]{
   GP1:
	UF : 1, UT : 5,		CONFIG : 'N U T, 0, 0, 0',
	X =  175.000  mm,	Y =  28.000  mm,	Z =   15.000 mm,
	W =-180.000 deg,	P =   0.000 deg,	R =    90.000 deg
};
P[2071]{
   GP1:
	UF : 1, UT : 5,		CONFIG : 'N U T, 0, 0, 0',
	X =  124.000  mm,	Y =  31.000  mm,	Z =   15.000 mm,
	W =-180.000 deg,	P =   0.000 deg,	R =    90.000 deg
};
P[2072]{
   GP1:
	UF : 1, UT : 5,		CONFIG : 'N U T, 0, 0, 0',
	X =  124.000  mm,	Y =  31.000  mm,	Z =   -1.000 mm,
	W =-180.000 deg,	P =   0.000 deg,	R =    90.000 deg
};
P[2073]{
   GP1:
	UF : 1, UT : 5,		CONFIG : 'N U T, 0, 0, 0',
	X =  124.000  mm,	Y =  31.000  mm,	Z =   15.000 mm,
	W =-180.000 deg,	P =   0.000 deg,	R =    90.000 deg
};
P[2083]{
   GP1:
	UF : 1, UT : 5,		CONFIG : 'N U T, 0, 0, 0',
	X =  136.000  mm,	Y =  31.000  mm,	Z =   15.000 mm,
	W =-180.000 deg,	P =   0.000 deg,	R =    90.000 deg
};
P[2084]{
   GP1:
	UF : 1, UT : 5,		CONFIG : 'N U T, 0, 0, 0',
	X =  136.000  mm,	Y =  31.000  mm,	Z =   -1.000 mm,
	W =-180.000 deg,	P =   0.000 deg,	R =    90.000 deg
};
P[2085]{
   GP1:
	UF : 1, UT : 5,		CONFIG : 'N U T, 0, 0, 0',
	X =  136.000  mm,	Y =  31.000  mm,	Z =   15.000 mm,
	W =-180.000 deg,	P =   0.000 deg,	R =    90.000 deg
};
P[2092]{
   GP1:
	UF : 1, UT : 5,		CONFIG : 'N U T, 0, 0, 0',
	X =  172.000  mm,	Y =  31.000  mm,	Z =   15.000 mm,
	W =-180.000 deg,	P =   0.000 deg,	R =    90.000 deg
};
P[2093]{
   GP1:
	UF : 1, UT : 5,		CONFIG : 'N U T, 0, 0, 0',
	X =  172.000  mm,	Y =  31.000  mm,	Z =   -1.000 mm,
	W =-180.000 deg,	P =   0.000 deg,	R =    90.000 deg
};
P[2094]{
   GP1:
	UF : 1, UT : 5,		CONFIG : 'N U T, 0, 0, 0',
	X =  172.000  mm,	Y =  31.000  mm,	Z =   15.000 mm,
	W =-180.000 deg,	P =   0.000 deg,	R =    90.000 deg
};
P[2116]{
   GP1:
	UF : 1, UT : 5,		CONFIG : 'N U T, 0, 0, 0',
	X =  16.000  mm,	Y =  34.000  mm,	Z =   15.000 mm,
	W =-180.000 deg,	P =   0.000 deg,	R =    90.000 deg
};
P[2117]{
   GP1:
	UF : 1, UT : 5,		CONFIG : 'N U T, 0, 0, 0',
	X =  16.000  mm,	Y =  34.000  mm,	Z =   -1.000 mm,
	W =-180.000 deg,	P =   0.000 deg,	R =    90.000 deg
};
P[2118]{
   GP1:
	UF : 1, UT : 5,		CONFIG : 'N U T, 0, 0, 0',
	X =  16.000  mm,	Y =  34.000  mm,	Z =   15.000 mm,
	W =-180.000 deg,	P =   0.000 deg,	R =    90.000 deg
};
P[2215]{
   GP1:
	UF : 1, UT : 5,		CONFIG : 'N U T, 0, 0, 0',
	X =  115.000  mm,	Y =  34.000  mm,	Z =   15.000 mm,
	W =-180.000 deg,	P =   0.000 deg,	R =    90.000 deg
};
P[2216]{
   GP1:
	UF : 1, UT : 5,		CONFIG : 'N U T, 0, 0, 0',
	X =  115.000  mm,	Y =  34.000  mm,	Z =   -1.000 mm,
	W =-180.000 deg,	P =   0.000 deg,	R =    90.000 deg
};
P[2217]{
   GP1:
	UF : 1, UT : 5,		CONFIG : 'N U T, 0, 0, 0',
	X =  115.000  mm,	Y =  34.000  mm,	Z =   15.000 mm,
	W =-180.000 deg,	P =   0.000 deg,	R =    90.000 deg
};
P[2221]{
   GP1:
	UF : 1, UT : 5,		CONFIG : 'N U T, 0, 0, 0',
	X =  121.000  mm,	Y =  34.000  mm,	Z =   15.000 mm,
	W =-180.000 deg,	P =   0.000 deg,	R =    90.000 deg
};
P[2222]{
   GP1:
	UF : 1, UT : 5,		CONFIG : 'N U T, 0, 0, 0',
	X =  121.000  mm,	Y =  34.000  mm,	Z =   -1.000 mm,
	W =-180.000 deg,	P =   0.000 deg,	R =    90.000 deg
};
P[2223]{
   GP1:
	UF : 1, UT : 5,		CONFIG : 'N U T, 0, 0, 0',
	X =  121.000  mm,	Y =  34.000  mm,	Z =   15.000 mm,
	W =-180.000 deg,	P =   0.000 deg,	R =    90.000 deg
};
P[2248]{
   GP1:
	UF : 1, UT : 5,		CONFIG : 'N U T, 0, 0, 0',
	X =  172.000  mm,	Y =  34.000  mm,	Z =   15.000 mm,
	W =-180.000 deg,	P =   0.000 deg,	R =    90.000 deg
};
P[2249]{
   GP1:
	UF : 1, UT : 5,		CONFIG : 'N U T, 0, 0, 0',
	X =  172.000  mm,	Y =  34.000  mm,	Z =   -1.000 mm,
	W =-180.000 deg,	P =   0.000 deg,	R =    90.000 deg
};
P[2250]{
   GP1:
	UF : 1, UT : 5,		CONFIG : 'N U T, 0, 0, 0',
	X =  172.000  mm,	Y =  34.000  mm,	Z =   15.000 mm,
	W =-180.000 deg,	P =   0.000 deg,	R =    90.000 deg
};
P[2509]{
   GP1:
	UF : 1, UT : 5,		CONFIG : 'N U T, 0, 0, 0',
	X =  118.000  mm,	Y =  40.000  mm,	Z =   15.000 mm,
	W =-180.000 deg,	P =   0.000 deg,	R =    90.000 deg
};
P[2510]{
   GP1:
	UF : 1, UT : 5,		CONFIG : 'N U T, 0, 0, 0',
	X =  118.000  mm,	Y =  40.000  mm,	Z =   -1.000 mm,
	W =-180.000 deg,	P =   0.000 deg,	R =    90.000 deg
};
P[2511]{
   GP1:
	UF : 1, UT : 5,		CONFIG : 'N U T, 0, 0, 0',
	X =  118.000  mm,	Y =  40.000  mm,	Z =   15.000 mm,
	W =-180.000 deg,	P =   0.000 deg,	R =    90.000 deg
};
P[2530]{
   GP1:
	UF : 1, UT : 5,		CONFIG : 'N U T, 0, 0, 0',
	X =  142.000  mm,	Y =  40.000  mm,	Z =   15.000 mm,
	W =-180.000 deg,	P =   0.000 deg,	R =    90.000 deg
};
P[2531]{
   GP1:
	UF : 1, UT : 5,		CONFIG : 'N U T, 0, 0, 0',
	X =  142.000  mm,	Y =  40.000  mm,	Z =   -1.000 mm,
	W =-180.000 deg,	P =   0.000 deg,	R =    90.000 deg
};
P[2532]{
   GP1:
	UF : 1, UT : 5,		CONFIG : 'N U T, 0, 0, 0',
	X =  142.000  mm,	Y =  40.000  mm,	Z =   15.000 mm,
	W =-180.000 deg,	P =   0.000 deg,	R =    90.000 deg
};
P[2650]{
   GP1:
	UF : 1, UT : 5,		CONFIG : 'N U T, 0, 0, 0',
	X =  124.000  mm,	Y =  43.000  mm,	Z =   15.000 mm,
	W =-180.000 deg,	P =   0.000 deg,	R =    90.000 deg
};
P[2651]{
   GP1:
	UF : 1, UT : 5,		CONFIG : 'N U T, 0, 0, 0',
	X =  124.000  mm,	Y =  43.000  mm,	Z =   -1.000 mm,
	W =-180.000 deg,	P =   0.000 deg,	R =    90.000 deg
};
P[2652]{
   GP1:
	UF : 1, UT : 5,		CONFIG : 'N U T, 0, 0, 0',
	X =  124.000  mm,	Y =  43.000  mm,	Z =   15.000 mm,
	W =-180.000 deg,	P =   0.000 deg,	R =    90.000 deg
};
P[2791]{
   GP1:
	UF : 1, UT : 5,		CONFIG : 'N U T, 0, 0, 0',
	X =  124.000  mm,	Y =  46.000  mm,	Z =   15.000 mm,
	W =-180.000 deg,	P =   0.000 deg,	R =    90.000 deg
};
P[2792]{
   GP1:
	UF : 1, UT : 5,		CONFIG : 'N U T, 0, 0, 0',
	X =  124.000  mm,	Y =  46.000  mm,	Z =   -1.000 mm,
	W =-180.000 deg,	P =   0.000 deg,	R =    90.000 deg
};
P[2793]{
   GP1:
	UF : 1, UT : 5,		CONFIG : 'N U T, 0, 0, 0',
	X =  124.000  mm,	Y =  46.000  mm,	Z =   15.000 mm,
	W =-180.000 deg,	P =   0.000 deg,	R =    90.000 deg
};
P[2809]{
   GP1:
	UF : 1, UT : 5,		CONFIG : 'N U T, 0, 0, 0',
	X =  142.000  mm,	Y =  46.000  mm,	Z =   15.000 mm,
	W =-180.000 deg,	P =   0.000 deg,	R =    90.000 deg
};
P[2810]{
   GP1:
	UF : 1, UT : 5,		CONFIG : 'N U T, 0, 0, 0',
	X =  142.000  mm,	Y =  46.000  mm,	Z =   -1.000 mm,
	W =-180.000 deg,	P =   0.000 deg,	R =    90.000 deg
};
P[2811]{
   GP1:
	UF : 1, UT : 5,		CONFIG : 'N U T, 0, 0, 0',
	X =  142.000  mm,	Y =  46.000  mm,	Z =   15.000 mm,
	W =-180.000 deg,	P =   0.000 deg,	R =    90.000 deg
};
P[2815]{
   GP1:
	UF : 1, UT : 5,		CONFIG : 'N U T, 0, 0, 0',
	X =  148.000  mm,	Y =  46.000  mm,	Z =   15.000 mm,
	W =-180.000 deg,	P =   0.000 deg,	R =    90.000 deg
};
P[2816]{
   GP1:
	UF : 1, UT : 5,		CONFIG : 'N U T, 0, 0, 0',
	X =  148.000  mm,	Y =  46.000  mm,	Z =   -1.000 mm,
	W =-180.000 deg,	P =   0.000 deg,	R =    90.000 deg
};
P[2817]{
   GP1:
	UF : 1, UT : 5,		CONFIG : 'N U T, 0, 0, 0',
	X =  148.000  mm,	Y =  46.000  mm,	Z =   15.000 mm,
	W =-180.000 deg,	P =   0.000 deg,	R =    90.000 deg
};
P[2818]{
   GP1:
	UF : 1, UT : 5,		CONFIG : 'N U T, 0, 0, 0',
	X =  154.000  mm,	Y =  46.000  mm,	Z =   15.000 mm,
	W =-180.000 deg,	P =   0.000 deg,	R =    90.000 deg
};
P[2819]{
   GP1:
	UF : 1, UT : 5,		CONFIG : 'N U T, 0, 0, 0',
	X =  154.000  mm,	Y =  46.000  mm,	Z =   -1.000 mm,
	W =-180.000 deg,	P =   0.000 deg,	R =    90.000 deg
};
P[2820]{
   GP1:
	UF : 1, UT : 5,		CONFIG : 'N U T, 0, 0, 0',
	X =  154.000  mm,	Y =  46.000  mm,	Z =   15.000 mm,
	W =-180.000 deg,	P =   0.000 deg,	R =    90.000 deg
};
P[2947]{
   GP1:
	UF : 1, UT : 5,		CONFIG : 'N U T, 0, 0, 0',
	X =  124.000  mm,	Y =  49.000  mm,	Z =   15.000 mm,
	W =-180.000 deg,	P =   0.000 deg,	R =    90.000 deg
};
P[2948]{
   GP1:
	UF : 1, UT : 5,		CONFIG : 'N U T, 0, 0, 0',
	X =  124.000  mm,	Y =  49.000  mm,	Z =   -1.000 mm,
	W =-180.000 deg,	P =   0.000 deg,	R =    90.000 deg
};
P[2949]{
   GP1:
	UF : 1, UT : 5,		CONFIG : 'N U T, 0, 0, 0',
	X =  124.000  mm,	Y =  49.000  mm,	Z =   15.000 mm,
	W =-180.000 deg,	P =   0.000 deg,	R =    90.000 deg
};
P[2956]{
   GP1:
	UF : 1, UT : 5,		CONFIG : 'N U T, 0, 0, 0',
	X =  133.000  mm,	Y =  49.000  mm,	Z =   15.000 mm,
	W =-180.000 deg,	P =   0.000 deg,	R =    90.000 deg
};
P[2957]{
   GP1:
	UF : 1, UT : 5,		CONFIG : 'N U T, 0, 0, 0',
	X =  133.000  mm,	Y =  49.000  mm,	Z =   -1.000 mm,
	W =-180.000 deg,	P =   0.000 deg,	R =    90.000 deg
};
P[2958]{
   GP1:
	UF : 1, UT : 5,		CONFIG : 'N U T, 0, 0, 0',
	X =  133.000  mm,	Y =  49.000  mm,	Z =   15.000 mm,
	W =-180.000 deg,	P =   0.000 deg,	R =    90.000 deg
};
P[2968]{
   GP1:
	UF : 1, UT : 5,		CONFIG : 'N U T, 0, 0, 0',
	X =  145.000  mm,	Y =  49.000  mm,	Z =   15.000 mm,
	W =-180.000 deg,	P =   0.000 deg,	R =    90.000 deg
};
P[2969]{
   GP1:
	UF : 1, UT : 5,		CONFIG : 'N U T, 0, 0, 0',
	X =  145.000  mm,	Y =  49.000  mm,	Z =   -1.000 mm,
	W =-180.000 deg,	P =   0.000 deg,	R =    90.000 deg
};
P[2970]{
   GP1:
	UF : 1, UT : 5,		CONFIG : 'N U T, 0, 0, 0',
	X =  145.000  mm,	Y =  49.000  mm,	Z =   15.000 mm,
	W =-180.000 deg,	P =   0.000 deg,	R =    90.000 deg
};
P[2971]{
   GP1:
	UF : 1, UT : 5,		CONFIG : 'N U T, 0, 0, 0',
	X =  148.000  mm,	Y =  49.000  mm,	Z =   15.000 mm,
	W =-180.000 deg,	P =   0.000 deg,	R =    90.000 deg
};
P[2972]{
   GP1:
	UF : 1, UT : 5,		CONFIG : 'N U T, 0, 0, 0',
	X =  148.000  mm,	Y =  49.000  mm,	Z =   -1.000 mm,
	W =-180.000 deg,	P =   0.000 deg,	R =    90.000 deg
};
P[2973]{
   GP1:
	UF : 1, UT : 5,		CONFIG : 'N U T, 0, 0, 0',
	X =  148.000  mm,	Y =  49.000  mm,	Z =   15.000 mm,
	W =-180.000 deg,	P =   0.000 deg,	R =    90.000 deg
};
P[2974]{
   GP1:
	UF : 1, UT : 5,		CONFIG : 'N U T, 0, 0, 0',
	X =  151.000  mm,	Y =  49.000  mm,	Z =   15.000 mm,
	W =-180.000 deg,	P =   0.000 deg,	R =    90.000 deg
};
P[2975]{
   GP1:
	UF : 1, UT : 5,		CONFIG : 'N U T, 0, 0, 0',
	X =  151.000  mm,	Y =  49.000  mm,	Z =   -1.000 mm,
	W =-180.000 deg,	P =   0.000 deg,	R =    90.000 deg
};
P[2976]{
   GP1:
	UF : 1, UT : 5,		CONFIG : 'N U T, 0, 0, 0',
	X =  151.000  mm,	Y =  49.000  mm,	Z =   15.000 mm,
	W =-180.000 deg,	P =   0.000 deg,	R =    90.000 deg
};
P[2977]{
   GP1:
	UF : 1, UT : 5,		CONFIG : 'N U T, 0, 0, 0',
	X =  154.000  mm,	Y =  49.000  mm,	Z =   15.000 mm,
	W =-180.000 deg,	P =   0.000 deg,	R =    90.000 deg
};
P[2978]{
   GP1:
	UF : 1, UT : 5,		CONFIG : 'N U T, 0, 0, 0',
	X =  154.000  mm,	Y =  49.000  mm,	Z =   -1.000 mm,
	W =-180.000 deg,	P =   0.000 deg,	R =    90.000 deg
};
P[2979]{
   GP1:
	UF : 1, UT : 5,		CONFIG : 'N U T, 0, 0, 0',
	X =  154.000  mm,	Y =  49.000  mm,	Z =   15.000 mm,
	W =-180.000 deg,	P =   0.000 deg,	R =    90.000 deg
};
P[3103]{
   GP1:
	UF : 1, UT : 5,		CONFIG : 'N U T, 0, 0, 0',
	X =  124.000  mm,	Y =  52.000  mm,	Z =   15.000 mm,
	W =-180.000 deg,	P =   0.000 deg,	R =    90.000 deg
};
P[3104]{
   GP1:
	UF : 1, UT : 5,		CONFIG : 'N U T, 0, 0, 0',
	X =  124.000  mm,	Y =  52.000  mm,	Z =   -1.000 mm,
	W =-180.000 deg,	P =   0.000 deg,	R =    90.000 deg
};
P[3105]{
   GP1:
	UF : 1, UT : 5,		CONFIG : 'N U T, 0, 0, 0',
	X =  124.000  mm,	Y =  52.000  mm,	Z =   15.000 mm,
	W =-180.000 deg,	P =   0.000 deg,	R =    90.000 deg
};
P[3109]{
   GP1:
	UF : 1, UT : 5,		CONFIG : 'N U T, 0, 0, 0',
	X =  130.000  mm,	Y =  52.000  mm,	Z =   15.000 mm,
	W =-180.000 deg,	P =   0.000 deg,	R =    90.000 deg
};
P[3110]{
   GP1:
	UF : 1, UT : 5,		CONFIG : 'N U T, 0, 0, 0',
	X =  130.000  mm,	Y =  52.000  mm,	Z =   -1.000 mm,
	W =-180.000 deg,	P =   0.000 deg,	R =    90.000 deg
};
P[3111]{
   GP1:
	UF : 1, UT : 5,		CONFIG : 'N U T, 0, 0, 0',
	X =  130.000  mm,	Y =  52.000  mm,	Z =   15.000 mm,
	W =-180.000 deg,	P =   0.000 deg,	R =    90.000 deg
};
P[3124]{
   GP1:
	UF : 1, UT : 5,		CONFIG : 'N U T, 0, 0, 0',
	X =  145.000  mm,	Y =  52.000  mm,	Z =   15.000 mm,
	W =-180.000 deg,	P =   0.000 deg,	R =    90.000 deg
};
P[3125]{
   GP1:
	UF : 1, UT : 5,		CONFIG : 'N U T, 0, 0, 0',
	X =  145.000  mm,	Y =  52.000  mm,	Z =   -1.000 mm,
	W =-180.000 deg,	P =   0.000 deg,	R =    90.000 deg
};
P[3126]{
   GP1:
	UF : 1, UT : 5,		CONFIG : 'N U T, 0, 0, 0',
	X =  145.000  mm,	Y =  52.000  mm,	Z =   15.000 mm,
	W =-180.000 deg,	P =   0.000 deg,	R =    90.000 deg
};
P[3127]{
   GP1:
	UF : 1, UT : 5,		CONFIG : 'N U T, 0, 0, 0',
	X =  148.000  mm,	Y =  52.000  mm,	Z =   15.000 mm,
	W =-180.000 deg,	P =   0.000 deg,	R =    90.000 deg
};
P[3128]{
   GP1:
	UF : 1, UT : 5,		CONFIG : 'N U T, 0, 0, 0',
	X =  148.000  mm,	Y =  52.000  mm,	Z =   -1.000 mm,
	W =-180.000 deg,	P =   0.000 deg,	R =    90.000 deg
};
P[3129]{
   GP1:
	UF : 1, UT : 5,		CONFIG : 'N U T, 0, 0, 0',
	X =  148.000  mm,	Y =  52.000  mm,	Z =   15.000 mm,
	W =-180.000 deg,	P =   0.000 deg,	R =    90.000 deg
};
P[3250]{
   GP1:
	UF : 1, UT : 5,		CONFIG : 'N U T, 0, 0, 0',
	X =  115.000  mm,	Y =  55.000  mm,	Z =   15.000 mm,
	W =-180.000 deg,	P =   0.000 deg,	R =    90.000 deg
};
P[3251]{
   GP1:
	UF : 1, UT : 5,		CONFIG : 'N U T, 0, 0, 0',
	X =  115.000  mm,	Y =  55.000  mm,	Z =   -1.000 mm,
	W =-180.000 deg,	P =   0.000 deg,	R =    90.000 deg
};
P[3252]{
   GP1:
	UF : 1, UT : 5,		CONFIG : 'N U T, 0, 0, 0',
	X =  115.000  mm,	Y =  55.000  mm,	Z =   15.000 mm,
	W =-180.000 deg,	P =   0.000 deg,	R =    90.000 deg
};
P[3253]{
   GP1:
	UF : 1, UT : 5,		CONFIG : 'N U T, 0, 0, 0',
	X =  121.000  mm,	Y =  55.000  mm,	Z =   15.000 mm,
	W =-180.000 deg,	P =   0.000 deg,	R =    90.000 deg
};
P[3254]{
   GP1:
	UF : 1, UT : 5,		CONFIG : 'N U T, 0, 0, 0',
	X =  121.000  mm,	Y =  55.000  mm,	Z =   -1.000 mm,
	W =-180.000 deg,	P =   0.000 deg,	R =    90.000 deg
};
P[3255]{
   GP1:
	UF : 1, UT : 5,		CONFIG : 'N U T, 0, 0, 0',
	X =  121.000  mm,	Y =  55.000  mm,	Z =   15.000 mm,
	W =-180.000 deg,	P =   0.000 deg,	R =    90.000 deg
};
P[3274]{
   GP1:
	UF : 1, UT : 5,		CONFIG : 'N U T, 0, 0, 0',
	X =  172.000  mm,	Y =  55.000  mm,	Z =   15.000 mm,
	W =-180.000 deg,	P =   0.000 deg,	R =    90.000 deg
};
P[3275]{
   GP1:
	UF : 1, UT : 5,		CONFIG : 'N U T, 0, 0, 0',
	X =  172.000  mm,	Y =  55.000  mm,	Z =   -1.000 mm,
	W =-180.000 deg,	P =   0.000 deg,	R =    90.000 deg
};
P[3276]{
   GP1:
	UF : 1, UT : 5,		CONFIG : 'N U T, 0, 0, 0',
	X =  172.000  mm,	Y =  55.000  mm,	Z =   15.000 mm,
	W =-180.000 deg,	P =   0.000 deg,	R =    90.000 deg
};
P[3403]{
   GP1:
	UF : 1, UT : 5,		CONFIG : 'N U T, 0, 0, 0',
	X =  130.000  mm,	Y =  58.000  mm,	Z =   15.000 mm,
	W =-180.000 deg,	P =   0.000 deg,	R =    90.000 deg
};
P[3404]{
   GP1:
	UF : 1, UT : 5,		CONFIG : 'N U T, 0, 0, 0',
	X =  130.000  mm,	Y =  58.000  mm,	Z =   -1.000 mm,
	W =-180.000 deg,	P =   0.000 deg,	R =    90.000 deg
};
P[3405]{
   GP1:
	UF : 1, UT : 5,		CONFIG : 'N U T, 0, 0, 0',
	X =  130.000  mm,	Y =  58.000  mm,	Z =   15.000 mm,
	W =-180.000 deg,	P =   0.000 deg,	R =    90.000 deg
};
P[3418]{
   GP1:
	UF : 1, UT : 5,		CONFIG : 'N U T, 0, 0, 0',
	X =  172.000  mm,	Y =  58.000  mm,	Z =   15.000 mm,
	W =-180.000 deg,	P =   0.000 deg,	R =    90.000 deg
};
P[3419]{
   GP1:
	UF : 1, UT : 5,		CONFIG : 'N U T, 0, 0, 0',
	X =  172.000  mm,	Y =  58.000  mm,	Z =   -1.000 mm,
	W =-180.000 deg,	P =   0.000 deg,	R =    90.000 deg
};
P[3420]{
   GP1:
	UF : 1, UT : 5,		CONFIG : 'N U T, 0, 0, 0',
	X =  172.000  mm,	Y =  58.000  mm,	Z =   15.000 mm,
	W =-180.000 deg,	P =   0.000 deg,	R =    90.000 deg
};
P[3541]{
   GP1:
	UF : 1, UT : 5,		CONFIG : 'N U T, 0, 0, 0',
	X =  124.000  mm,	Y =  61.000  mm,	Z =   15.000 mm,
	W =-180.000 deg,	P =   0.000 deg,	R =    90.000 deg
};
P[3542]{
   GP1:
	UF : 1, UT : 5,		CONFIG : 'N U T, 0, 0, 0',
	X =  124.000  mm,	Y =  61.000  mm,	Z =   -1.000 mm,
	W =-180.000 deg,	P =   0.000 deg,	R =    90.000 deg
};
P[3543]{
   GP1:
	UF : 1, UT : 5,		CONFIG : 'N U T, 0, 0, 0',
	X =  124.000  mm,	Y =  61.000  mm,	Z =   15.000 mm,
	W =-180.000 deg,	P =   0.000 deg,	R =    90.000 deg
};
P[3544]{
   GP1:
	UF : 1, UT : 5,		CONFIG : 'N U T, 0, 0, 0',
	X =  127.000  mm,	Y =  61.000  mm,	Z =   15.000 mm,
	W =-180.000 deg,	P =   0.000 deg,	R =    90.000 deg
};
P[3545]{
   GP1:
	UF : 1, UT : 5,		CONFIG : 'N U T, 0, 0, 0',
	X =  127.000  mm,	Y =  61.000  mm,	Z =   -1.000 mm,
	W =-180.000 deg,	P =   0.000 deg,	R =    90.000 deg
};
P[3546]{
   GP1:
	UF : 1, UT : 5,		CONFIG : 'N U T, 0, 0, 0',
	X =  127.000  mm,	Y =  61.000  mm,	Z =   15.000 mm,
	W =-180.000 deg,	P =   0.000 deg,	R =    90.000 deg
};
P[3547]{
   GP1:
	UF : 1, UT : 5,		CONFIG : 'N U T, 0, 0, 0',
	X =  130.000  mm,	Y =  61.000  mm,	Z =   15.000 mm,
	W =-180.000 deg,	P =   0.000 deg,	R =    90.000 deg
};
P[3548]{
   GP1:
	UF : 1, UT : 5,		CONFIG : 'N U T, 0, 0, 0',
	X =  130.000  mm,	Y =  61.000  mm,	Z =   -1.000 mm,
	W =-180.000 deg,	P =   0.000 deg,	R =    90.000 deg
};
P[3549]{
   GP1:
	UF : 1, UT : 5,		CONFIG : 'N U T, 0, 0, 0',
	X =  130.000  mm,	Y =  61.000  mm,	Z =   15.000 mm,
	W =-180.000 deg,	P =   0.000 deg,	R =    90.000 deg
};
P[3556]{
   GP1:
	UF : 1, UT : 5,		CONFIG : 'N U T, 0, 0, 0',
	X =  142.000  mm,	Y =  61.000  mm,	Z =   15.000 mm,
	W =-180.000 deg,	P =   0.000 deg,	R =    90.000 deg
};
P[3557]{
   GP1:
	UF : 1, UT : 5,		CONFIG : 'N U T, 0, 0, 0',
	X =  142.000  mm,	Y =  61.000  mm,	Z =   -1.000 mm,
	W =-180.000 deg,	P =   0.000 deg,	R =    90.000 deg
};
P[3558]{
   GP1:
	UF : 1, UT : 5,		CONFIG : 'N U T, 0, 0, 0',
	X =  142.000  mm,	Y =  61.000  mm,	Z =   15.000 mm,
	W =-180.000 deg,	P =   0.000 deg,	R =    90.000 deg
};
P[3700]{
   GP1:
	UF : 1, UT : 5,		CONFIG : 'N U T, 0, 0, 0',
	X =  139.000  mm,	Y =  64.000  mm,	Z =   15.000 mm,
	W =-180.000 deg,	P =   0.000 deg,	R =    90.000 deg
};
P[3701]{
   GP1:
	UF : 1, UT : 5,		CONFIG : 'N U T, 0, 0, 0',
	X =  139.000  mm,	Y =  64.000  mm,	Z =   -1.000 mm,
	W =-180.000 deg,	P =   0.000 deg,	R =    90.000 deg
};
P[3702]{
   GP1:
	UF : 1, UT : 5,		CONFIG : 'N U T, 0, 0, 0',
	X =  139.000  mm,	Y =  64.000  mm,	Z =   15.000 mm,
	W =-180.000 deg,	P =   0.000 deg,	R =    90.000 deg
};
P[3838]{
   GP1:
	UF : 1, UT : 5,		CONFIG : 'N U T, 0, 0, 0',
	X =  139.000  mm,	Y =  67.000  mm,	Z =   15.000 mm,
	W =-180.000 deg,	P =   0.000 deg,	R =    90.000 deg
};
P[3839]{
   GP1:
	UF : 1, UT : 5,		CONFIG : 'N U T, 0, 0, 0',
	X =  139.000  mm,	Y =  67.000  mm,	Z =   -1.000 mm,
	W =-180.000 deg,	P =   0.000 deg,	R =    90.000 deg
};
P[3840]{
   GP1:
	UF : 1, UT : 5,		CONFIG : 'N U T, 0, 0, 0',
	X =  139.000  mm,	Y =  67.000  mm,	Z =   15.000 mm,
	W =-180.000 deg,	P =   0.000 deg,	R =    90.000 deg
};
P[3973]{
   GP1:
	UF : 1, UT : 5,		CONFIG : 'N U T, 0, 0, 0',
	X =  136.000  mm,	Y =  70.000  mm,	Z =   15.000 mm,
	W =-180.000 deg,	P =   0.000 deg,	R =    90.000 deg
};
P[3974]{
   GP1:
	UF : 1, UT : 5,		CONFIG : 'N U T, 0, 0, 0',
	X =  136.000  mm,	Y =  70.000  mm,	Z =   -1.000 mm,
	W =-180.000 deg,	P =   0.000 deg,	R =    90.000 deg
};
P[3975]{
   GP1:
	UF : 1, UT : 5,		CONFIG : 'N U T, 0, 0, 0',
	X =  136.000  mm,	Y =  70.000  mm,	Z =   15.000 mm,
	W =-180.000 deg,	P =   0.000 deg,	R =    90.000 deg
};
P[3985]{
   GP1:
	UF : 1, UT : 5,		CONFIG : 'N U T, 0, 0, 0',
	X =  169.000  mm,	Y =  70.000  mm,	Z =   15.000 mm,
	W =-180.000 deg,	P =   0.000 deg,	R =    90.000 deg
};
P[3986]{
   GP1:
	UF : 1, UT : 5,		CONFIG : 'N U T, 0, 0, 0',
	X =  169.000  mm,	Y =  70.000  mm,	Z =   -1.000 mm,
	W =-180.000 deg,	P =   0.000 deg,	R =    90.000 deg
};
P[3987]{
   GP1:
	UF : 1, UT : 5,		CONFIG : 'N U T, 0, 0, 0',
	X =  169.000  mm,	Y =  70.000  mm,	Z =   15.000 mm,
	W =-180.000 deg,	P =   0.000 deg,	R =    90.000 deg
};
P[4009]{
   GP1:
	UF : 1, UT : 5,		CONFIG : 'N U T, 0, 0, 0',
	X =  13.000  mm,	Y =  73.000  mm,	Z =   15.000 mm,
	W =-180.000 deg,	P =   0.000 deg,	R =    90.000 deg
};
P[4010]{
   GP1:
	UF : 1, UT : 5,		CONFIG : 'N U T, 0, 0, 0',
	X =  13.000  mm,	Y =  73.000  mm,	Z =   -1.000 mm,
	W =-180.000 deg,	P =   0.000 deg,	R =    90.000 deg
};
P[4011]{
   GP1:
	UF : 1, UT : 5,		CONFIG : 'N U T, 0, 0, 0',
	X =  13.000  mm,	Y =  73.000  mm,	Z =   15.000 mm,
	W =-180.000 deg,	P =   0.000 deg,	R =    90.000 deg
};
P[4069]{
   GP1:
	UF : 1, UT : 5,		CONFIG : 'N U T, 0, 0, 0',
	X =  76.000  mm,	Y =  73.000  mm,	Z =   15.000 mm,
	W =-180.000 deg,	P =   0.000 deg,	R =    90.000 deg
};
P[4070]{
   GP1:
	UF : 1, UT : 5,		CONFIG : 'N U T, 0, 0, 0',
	X =  76.000  mm,	Y =  73.000  mm,	Z =   -1.000 mm,
	W =-180.000 deg,	P =   0.000 deg,	R =    90.000 deg
};
P[4071]{
   GP1:
	UF : 1, UT : 5,		CONFIG : 'N U T, 0, 0, 0',
	X =  76.000  mm,	Y =  73.000  mm,	Z =   15.000 mm,
	W =-180.000 deg,	P =   0.000 deg,	R =    90.000 deg
};
P[4291]{
   GP1:
	UF : 1, UT : 5,		CONFIG : 'N U T, 0, 0, 0',
	X =  34.000  mm,	Y =  79.000  mm,	Z =   15.000 mm,
	W =-180.000 deg,	P =   0.000 deg,	R =    90.000 deg
};
P[4292]{
   GP1:
	UF : 1, UT : 5,		CONFIG : 'N U T, 0, 0, 0',
	X =  34.000  mm,	Y =  79.000  mm,	Z =   -1.000 mm,
	W =-180.000 deg,	P =   0.000 deg,	R =    90.000 deg
};
P[4293]{
   GP1:
	UF : 1, UT : 5,		CONFIG : 'N U T, 0, 0, 0',
	X =  34.000  mm,	Y =  79.000  mm,	Z =   15.000 mm,
	W =-180.000 deg,	P =   0.000 deg,	R =    90.000 deg
};
P[4369]{
   GP1:
	UF : 1, UT : 5,		CONFIG : 'N U T, 0, 0, 0',
	X =  130.000  mm,	Y =  79.000  mm,	Z =   15.000 mm,
	W =-180.000 deg,	P =   0.000 deg,	R =    90.000 deg
};
P[4370]{
   GP1:
	UF : 1, UT : 5,		CONFIG : 'N U T, 0, 0, 0',
	X =  130.000  mm,	Y =  79.000  mm,	Z =   -1.000 mm,
	W =-180.000 deg,	P =   0.000 deg,	R =    90.000 deg
};
P[4371]{
   GP1:
	UF : 1, UT : 5,		CONFIG : 'N U T, 0, 0, 0',
	X =  130.000  mm,	Y =  79.000  mm,	Z =   15.000 mm,
	W =-180.000 deg,	P =   0.000 deg,	R =    90.000 deg
};
P[4510]{
   GP1:
	UF : 1, UT : 5,		CONFIG : 'N U T, 0, 0, 0',
	X =  130.000  mm,	Y =  82.000  mm,	Z =   15.000 mm,
	W =-180.000 deg,	P =   0.000 deg,	R =    90.000 deg
};
P[4511]{
   GP1:
	UF : 1, UT : 5,		CONFIG : 'N U T, 0, 0, 0',
	X =  130.000  mm,	Y =  82.000  mm,	Z =   -1.000 mm,
	W =-180.000 deg,	P =   0.000 deg,	R =    90.000 deg
};
P[4512]{
   GP1:
	UF : 1, UT : 5,		CONFIG : 'N U T, 0, 0, 0',
	X =  130.000  mm,	Y =  82.000  mm,	Z =   15.000 mm,
	W =-180.000 deg,	P =   0.000 deg,	R =    90.000 deg
};
P[4519]{
   GP1:
	UF : 1, UT : 5,		CONFIG : 'N U T, 0, 0, 0',
	X =  139.000  mm,	Y =  82.000  mm,	Z =   15.000 mm,
	W =-180.000 deg,	P =   0.000 deg,	R =    90.000 deg
};
P[4520]{
   GP1:
	UF : 1, UT : 5,		CONFIG : 'N U T, 0, 0, 0',
	X =  139.000  mm,	Y =  82.000  mm,	Z =   -1.000 mm,
	W =-180.000 deg,	P =   0.000 deg,	R =    90.000 deg
};
P[4521]{
   GP1:
	UF : 1, UT : 5,		CONFIG : 'N U T, 0, 0, 0',
	X =  139.000  mm,	Y =  82.000  mm,	Z =   15.000 mm,
	W =-180.000 deg,	P =   0.000 deg,	R =    90.000 deg
};
P[4525]{
   GP1:
	UF : 1, UT : 5,		CONFIG : 'N U T, 0, 0, 0',
	X =  145.000  mm,	Y =  82.000  mm,	Z =   15.000 mm,
	W =-180.000 deg,	P =   0.000 deg,	R =    90.000 deg
};
P[4526]{
   GP1:
	UF : 1, UT : 5,		CONFIG : 'N U T, 0, 0, 0',
	X =  145.000  mm,	Y =  82.000  mm,	Z =   -1.000 mm,
	W =-180.000 deg,	P =   0.000 deg,	R =    90.000 deg
};
P[4527]{
   GP1:
	UF : 1, UT : 5,		CONFIG : 'N U T, 0, 0, 0',
	X =  145.000  mm,	Y =  82.000  mm,	Z =   15.000 mm,
	W =-180.000 deg,	P =   0.000 deg,	R =    90.000 deg
};
P[4528]{
   GP1:
	UF : 1, UT : 5,		CONFIG : 'N U T, 0, 0, 0',
	X =  166.000  mm,	Y =  82.000  mm,	Z =   15.000 mm,
	W =-180.000 deg,	P =   0.000 deg,	R =    90.000 deg
};
P[4529]{
   GP1:
	UF : 1, UT : 5,		CONFIG : 'N U T, 0, 0, 0',
	X =  166.000  mm,	Y =  82.000  mm,	Z =   -1.000 mm,
	W =-180.000 deg,	P =   0.000 deg,	R =    90.000 deg
};
P[4530]{
   GP1:
	UF : 1, UT : 5,		CONFIG : 'N U T, 0, 0, 0',
	X =  166.000  mm,	Y =  82.000  mm,	Z =   15.000 mm,
	W =-180.000 deg,	P =   0.000 deg,	R =    90.000 deg
};
P[4657]{
   GP1:
	UF : 1, UT : 5,		CONFIG : 'N U T, 0, 0, 0',
	X =  127.000  mm,	Y =  85.000  mm,	Z =   15.000 mm,
	W =-180.000 deg,	P =   0.000 deg,	R =    90.000 deg
};
P[4658]{
   GP1:
	UF : 1, UT : 5,		CONFIG : 'N U T, 0, 0, 0',
	X =  127.000  mm,	Y =  85.000  mm,	Z =   -1.000 mm,
	W =-180.000 deg,	P =   0.000 deg,	R =    90.000 deg
};
P[4659]{
   GP1:
	UF : 1, UT : 5,		CONFIG : 'N U T, 0, 0, 0',
	X =  127.000  mm,	Y =  85.000  mm,	Z =   15.000 mm,
	W =-180.000 deg,	P =   0.000 deg,	R =    90.000 deg
};
P[4660]{
   GP1:
	UF : 1, UT : 5,		CONFIG : 'N U T, 0, 0, 0',
	X =  130.000  mm,	Y =  85.000  mm,	Z =   15.000 mm,
	W =-180.000 deg,	P =   0.000 deg,	R =    90.000 deg
};
P[4661]{
   GP1:
	UF : 1, UT : 5,		CONFIG : 'N U T, 0, 0, 0',
	X =  130.000  mm,	Y =  85.000  mm,	Z =   -1.000 mm,
	W =-180.000 deg,	P =   0.000 deg,	R =    90.000 deg
};
P[4662]{
   GP1:
	UF : 1, UT : 5,		CONFIG : 'N U T, 0, 0, 0',
	X =  130.000  mm,	Y =  85.000  mm,	Z =   15.000 mm,
	W =-180.000 deg,	P =   0.000 deg,	R =    90.000 deg
};
P[4807]{
   GP1:
	UF : 1, UT : 5,		CONFIG : 'N U T, 0, 0, 0',
	X =  118.000  mm,	Y =  88.000  mm,	Z =   15.000 mm,
	W =-180.000 deg,	P =   0.000 deg,	R =    90.000 deg
};
P[4808]{
   GP1:
	UF : 1, UT : 5,		CONFIG : 'N U T, 0, 0, 0',
	X =  118.000  mm,	Y =  88.000  mm,	Z =   -1.000 mm,
	W =-180.000 deg,	P =   0.000 deg,	R =    90.000 deg
};
P[4809]{
   GP1:
	UF : 1, UT : 5,		CONFIG : 'N U T, 0, 0, 0',
	X =  118.000  mm,	Y =  88.000  mm,	Z =   15.000 mm,
	W =-180.000 deg,	P =   0.000 deg,	R =    90.000 deg
};
P[4813]{
   GP1:
	UF : 1, UT : 5,		CONFIG : 'N U T, 0, 0, 0',
	X =  133.000  mm,	Y =  88.000  mm,	Z =   15.000 mm,
	W =-180.000 deg,	P =   0.000 deg,	R =    90.000 deg
};
P[4814]{
   GP1:
	UF : 1, UT : 5,		CONFIG : 'N U T, 0, 0, 0',
	X =  133.000  mm,	Y =  88.000  mm,	Z =   -1.000 mm,
	W =-180.000 deg,	P =   0.000 deg,	R =    90.000 deg
};
P[4815]{
   GP1:
	UF : 1, UT : 5,		CONFIG : 'N U T, 0, 0, 0',
	X =  133.000  mm,	Y =  88.000  mm,	Z =   15.000 mm,
	W =-180.000 deg,	P =   0.000 deg,	R =    90.000 deg
};
P[4819]{
   GP1:
	UF : 1, UT : 5,		CONFIG : 'N U T, 0, 0, 0',
	X =  139.000  mm,	Y =  88.000  mm,	Z =   15.000 mm,
	W =-180.000 deg,	P =   0.000 deg,	R =    90.000 deg
};
P[4820]{
   GP1:
	UF : 1, UT : 5,		CONFIG : 'N U T, 0, 0, 0',
	X =  139.000  mm,	Y =  88.000  mm,	Z =   -1.000 mm,
	W =-180.000 deg,	P =   0.000 deg,	R =    90.000 deg
};
P[4821]{
   GP1:
	UF : 1, UT : 5,		CONFIG : 'N U T, 0, 0, 0',
	X =  139.000  mm,	Y =  88.000  mm,	Z =   15.000 mm,
	W =-180.000 deg,	P =   0.000 deg,	R =    90.000 deg
};
P[4948]{
   GP1:
	UF : 1, UT : 5,		CONFIG : 'N U T, 0, 0, 0',
	X =  118.000  mm,	Y =  91.000  mm,	Z =   15.000 mm,
	W =-180.000 deg,	P =   0.000 deg,	R =    90.000 deg
};
P[4949]{
   GP1:
	UF : 1, UT : 5,		CONFIG : 'N U T, 0, 0, 0',
	X =  118.000  mm,	Y =  91.000  mm,	Z =   -1.000 mm,
	W =-180.000 deg,	P =   0.000 deg,	R =    90.000 deg
};
P[4950]{
   GP1:
	UF : 1, UT : 5,		CONFIG : 'N U T, 0, 0, 0',
	X =  118.000  mm,	Y =  91.000  mm,	Z =   15.000 mm,
	W =-180.000 deg,	P =   0.000 deg,	R =    90.000 deg
};
P[4951]{
   GP1:
	UF : 1, UT : 5,		CONFIG : 'N U T, 0, 0, 0',
	X =  121.000  mm,	Y =  91.000  mm,	Z =   15.000 mm,
	W =-180.000 deg,	P =   0.000 deg,	R =    90.000 deg
};
P[4952]{
   GP1:
	UF : 1, UT : 5,		CONFIG : 'N U T, 0, 0, 0',
	X =  121.000  mm,	Y =  91.000  mm,	Z =   -1.000 mm,
	W =-180.000 deg,	P =   0.000 deg,	R =    90.000 deg
};
P[4953]{
   GP1:
	UF : 1, UT : 5,		CONFIG : 'N U T, 0, 0, 0',
	X =  121.000  mm,	Y =  91.000  mm,	Z =   15.000 mm,
	W =-180.000 deg,	P =   0.000 deg,	R =    90.000 deg
};
P[4954]{
   GP1:
	UF : 1, UT : 5,		CONFIG : 'N U T, 0, 0, 0',
	X =  124.000  mm,	Y =  91.000  mm,	Z =   15.000 mm,
	W =-180.000 deg,	P =   0.000 deg,	R =    90.000 deg
};
P[4955]{
   GP1:
	UF : 1, UT : 5,		CONFIG : 'N U T, 0, 0, 0',
	X =  124.000  mm,	Y =  91.000  mm,	Z =   -1.000 mm,
	W =-180.000 deg,	P =   0.000 deg,	R =    90.000 deg
};
P[4956]{
   GP1:
	UF : 1, UT : 5,		CONFIG : 'N U T, 0, 0, 0',
	X =  124.000  mm,	Y =  91.000  mm,	Z =   15.000 mm,
	W =-180.000 deg,	P =   0.000 deg,	R =    90.000 deg
};
P[4957]{
   GP1:
	UF : 1, UT : 5,		CONFIG : 'N U T, 0, 0, 0',
	X =  130.000  mm,	Y =  91.000  mm,	Z =   15.000 mm,
	W =-180.000 deg,	P =   0.000 deg,	R =    90.000 deg
};
P[4958]{
   GP1:
	UF : 1, UT : 5,		CONFIG : 'N U T, 0, 0, 0',
	X =  130.000  mm,	Y =  91.000  mm,	Z =   -1.000 mm,
	W =-180.000 deg,	P =   0.000 deg,	R =    90.000 deg
};
P[4959]{
   GP1:
	UF : 1, UT : 5,		CONFIG : 'N U T, 0, 0, 0',
	X =  130.000  mm,	Y =  91.000  mm,	Z =   15.000 mm,
	W =-180.000 deg,	P =   0.000 deg,	R =    90.000 deg
};
P[5110]{
   GP1:
	UF : 1, UT : 5,		CONFIG : 'N U T, 0, 0, 0',
	X =  163.000  mm,	Y =  94.000  mm,	Z =   15.000 mm,
	W =-180.000 deg,	P =   0.000 deg,	R =    90.000 deg
};
P[5111]{
   GP1:
	UF : 1, UT : 5,		CONFIG : 'N U T, 0, 0, 0',
	X =  163.000  mm,	Y =  94.000  mm,	Z =   -1.000 mm,
	W =-180.000 deg,	P =   0.000 deg,	R =    90.000 deg
};
P[5112]{
   GP1:
	UF : 1, UT : 5,		CONFIG : 'N U T, 0, 0, 0',
	X =  163.000  mm,	Y =  94.000  mm,	Z =   15.000 mm,
	W =-180.000 deg,	P =   0.000 deg,	R =    90.000 deg
};
P[5248]{
   GP1:
	UF : 1, UT : 5,		CONFIG : 'N U T, 0, 0, 0',
	X =  121.000  mm,	Y =  97.000  mm,	Z =   15.000 mm,
	W =-180.000 deg,	P =   0.000 deg,	R =    90.000 deg
};
P[5249]{
   GP1:
	UF : 1, UT : 5,		CONFIG : 'N U T, 0, 0, 0',
	X =  121.000  mm,	Y =  97.000  mm,	Z =   -1.000 mm,
	W =-180.000 deg,	P =   0.000 deg,	R =    90.000 deg
};
P[5250]{
   GP1:
	UF : 1, UT : 5,		CONFIG : 'N U T, 0, 0, 0',
	X =  121.000  mm,	Y =  97.000  mm,	Z =   15.000 mm,
	W =-180.000 deg,	P =   0.000 deg,	R =    90.000 deg
};
P[5251]{
   GP1:
	UF : 1, UT : 5,		CONFIG : 'N U T, 0, 0, 0',
	X =  124.000  mm,	Y =  97.000  mm,	Z =   15.000 mm,
	W =-180.000 deg,	P =   0.000 deg,	R =    90.000 deg
};
P[5252]{
   GP1:
	UF : 1, UT : 5,		CONFIG : 'N U T, 0, 0, 0',
	X =  124.000  mm,	Y =  97.000  mm,	Z =   -1.000 mm,
	W =-180.000 deg,	P =   0.000 deg,	R =    90.000 deg
};
P[5253]{
   GP1:
	UF : 1, UT : 5,		CONFIG : 'N U T, 0, 0, 0',
	X =  124.000  mm,	Y =  97.000  mm,	Z =   15.000 mm,
	W =-180.000 deg,	P =   0.000 deg,	R =    90.000 deg
};
P[5257]{
   GP1:
	UF : 1, UT : 5,		CONFIG : 'N U T, 0, 0, 0',
	X =  130.000  mm,	Y =  97.000  mm,	Z =   15.000 mm,
	W =-180.000 deg,	P =   0.000 deg,	R =    90.000 deg
};
P[5258]{
   GP1:
	UF : 1, UT : 5,		CONFIG : 'N U T, 0, 0, 0',
	X =  130.000  mm,	Y =  97.000  mm,	Z =   -1.000 mm,
	W =-180.000 deg,	P =   0.000 deg,	R =    90.000 deg
};
P[5259]{
   GP1:
	UF : 1, UT : 5,		CONFIG : 'N U T, 0, 0, 0',
	X =  130.000  mm,	Y =  97.000  mm,	Z =   15.000 mm,
	W =-180.000 deg,	P =   0.000 deg,	R =    90.000 deg
};
P[5422]{
   GP1:
	UF : 1, UT : 5,		CONFIG : 'N U T, 0, 0, 0',
	X =  127.000  mm,	Y =  100.000  mm,	Z =   15.000 mm,
	W =-180.000 deg,	P =   0.000 deg,	R =    90.000 deg
};
P[5423]{
   GP1:
	UF : 1, UT : 5,		CONFIG : 'N U T, 0, 0, 0',
	X =  127.000  mm,	Y =  100.000  mm,	Z =   -1.000 mm,
	W =-180.000 deg,	P =   0.000 deg,	R =    90.000 deg
};
P[5424]{
   GP1:
	UF : 1, UT : 5,		CONFIG : 'N U T, 0, 0, 0',
	X =  127.000  mm,	Y =  100.000  mm,	Z =   15.000 mm,
	W =-180.000 deg,	P =   0.000 deg,	R =    90.000 deg
};
P[5425]{
   GP1:
	UF : 1, UT : 5,		CONFIG : 'N U T, 0, 0, 0',
	X =  130.000  mm,	Y =  100.000  mm,	Z =   15.000 mm,
	W =-180.000 deg,	P =   0.000 deg,	R =    90.000 deg
};
P[5426]{
   GP1:
	UF : 1, UT : 5,		CONFIG : 'N U T, 0, 0, 0',
	X =  130.000  mm,	Y =  100.000  mm,	Z =   -1.000 mm,
	W =-180.000 deg,	P =   0.000 deg,	R =    90.000 deg
};
P[5427]{
   GP1:
	UF : 1, UT : 5,		CONFIG : 'N U T, 0, 0, 0',
	X =  130.000  mm,	Y =  100.000  mm,	Z =   15.000 mm,
	W =-180.000 deg,	P =   0.000 deg,	R =    90.000 deg
};
P[5584]{
   GP1:
	UF : 1, UT : 5,		CONFIG : 'N U T, 0, 0, 0',
	X =  121.000  mm,	Y =  103.000  mm,	Z =   15.000 mm,
	W =-180.000 deg,	P =   0.000 deg,	R =    90.000 deg
};
P[5585]{
   GP1:
	UF : 1, UT : 5,		CONFIG : 'N U T, 0, 0, 0',
	X =  121.000  mm,	Y =  103.000  mm,	Z =   -1.000 mm,
	W =-180.000 deg,	P =   0.000 deg,	R =    90.000 deg
};
P[5586]{
   GP1:
	UF : 1, UT : 5,		CONFIG : 'N U T, 0, 0, 0',
	X =  121.000  mm,	Y =  103.000  mm,	Z =   15.000 mm,
	W =-180.000 deg,	P =   0.000 deg,	R =    90.000 deg
};
P[5587]{
   GP1:
	UF : 1, UT : 5,		CONFIG : 'N U T, 0, 0, 0',
	X =  124.000  mm,	Y =  103.000  mm,	Z =   15.000 mm,
	W =-180.000 deg,	P =   0.000 deg,	R =    90.000 deg
};
P[5588]{
   GP1:
	UF : 1, UT : 5,		CONFIG : 'N U T, 0, 0, 0',
	X =  124.000  mm,	Y =  103.000  mm,	Z =   -1.000 mm,
	W =-180.000 deg,	P =   0.000 deg,	R =    90.000 deg
};
P[5589]{
   GP1:
	UF : 1, UT : 5,		CONFIG : 'N U T, 0, 0, 0',
	X =  124.000  mm,	Y =  103.000  mm,	Z =   15.000 mm,
	W =-180.000 deg,	P =   0.000 deg,	R =    90.000 deg
};
P[5590]{
   GP1:
	UF : 1, UT : 5,		CONFIG : 'N U T, 0, 0, 0',
	X =  127.000  mm,	Y =  103.000  mm,	Z =   15.000 mm,
	W =-180.000 deg,	P =   0.000 deg,	R =    90.000 deg
};
P[5591]{
   GP1:
	UF : 1, UT : 5,		CONFIG : 'N U T, 0, 0, 0',
	X =  127.000  mm,	Y =  103.000  mm,	Z =   -1.000 mm,
	W =-180.000 deg,	P =   0.000 deg,	R =    90.000 deg
};
P[5592]{
   GP1:
	UF : 1, UT : 5,		CONFIG : 'N U T, 0, 0, 0',
	X =  127.000  mm,	Y =  103.000  mm,	Z =   15.000 mm,
	W =-180.000 deg,	P =   0.000 deg,	R =    90.000 deg
};
P[5593]{
   GP1:
	UF : 1, UT : 5,		CONFIG : 'N U T, 0, 0, 0',
	X =  130.000  mm,	Y =  103.000  mm,	Z =   15.000 mm,
	W =-180.000 deg,	P =   0.000 deg,	R =    90.000 deg
};
P[5594]{
   GP1:
	UF : 1, UT : 5,		CONFIG : 'N U T, 0, 0, 0',
	X =  130.000  mm,	Y =  103.000  mm,	Z =   -1.000 mm,
	W =-180.000 deg,	P =   0.000 deg,	R =    90.000 deg
};
P[5595]{
   GP1:
	UF : 1, UT : 5,		CONFIG : 'N U T, 0, 0, 0',
	X =  130.000  mm,	Y =  103.000  mm,	Z =   15.000 mm,
	W =-180.000 deg,	P =   0.000 deg,	R =    90.000 deg
};
P[5599]{
   GP1:
	UF : 1, UT : 5,		CONFIG : 'N U T, 0, 0, 0',
	X =  136.000  mm,	Y =  103.000  mm,	Z =   15.000 mm,
	W =-180.000 deg,	P =   0.000 deg,	R =    90.000 deg
};
P[5600]{
   GP1:
	UF : 1, UT : 5,		CONFIG : 'N U T, 0, 0, 0',
	X =  136.000  mm,	Y =  103.000  mm,	Z =   -1.000 mm,
	W =-180.000 deg,	P =   0.000 deg,	R =    90.000 deg
};
P[5601]{
   GP1:
	UF : 1, UT : 5,		CONFIG : 'N U T, 0, 0, 0',
	X =  136.000  mm,	Y =  103.000  mm,	Z =   15.000 mm,
	W =-180.000 deg,	P =   0.000 deg,	R =    90.000 deg
};
P[5611]{
   GP1:
	UF : 1, UT : 5,		CONFIG : 'N U T, 0, 0, 0',
	X =  148.000  mm,	Y =  103.000  mm,	Z =   15.000 mm,
	W =-180.000 deg,	P =   0.000 deg,	R =    90.000 deg
};
P[5612]{
   GP1:
	UF : 1, UT : 5,		CONFIG : 'N U T, 0, 0, 0',
	X =  148.000  mm,	Y =  103.000  mm,	Z =   -1.000 mm,
	W =-180.000 deg,	P =   0.000 deg,	R =    90.000 deg
};
P[5613]{
   GP1:
	UF : 1, UT : 5,		CONFIG : 'N U T, 0, 0, 0',
	X =  148.000  mm,	Y =  103.000  mm,	Z =   15.000 mm,
	W =-180.000 deg,	P =   0.000 deg,	R =    90.000 deg
};
P[5614]{
   GP1:
	UF : 1, UT : 5,		CONFIG : 'N U T, 0, 0, 0',
	X =  160.000  mm,	Y =  103.000  mm,	Z =   15.000 mm,
	W =-180.000 deg,	P =   0.000 deg,	R =    90.000 deg
};
P[5615]{
   GP1:
	UF : 1, UT : 5,		CONFIG : 'N U T, 0, 0, 0',
	X =  160.000  mm,	Y =  103.000  mm,	Z =   -1.000 mm,
	W =-180.000 deg,	P =   0.000 deg,	R =    90.000 deg
};
P[5616]{
   GP1:
	UF : 1, UT : 5,		CONFIG : 'N U T, 0, 0, 0',
	X =  160.000  mm,	Y =  103.000  mm,	Z =   15.000 mm,
	W =-180.000 deg,	P =   0.000 deg,	R =    90.000 deg
};
P[5689]{
   GP1:
	UF : 1, UT : 5,		CONFIG : 'N U T, 0, 0, 0',
	X =  55.000  mm,	Y =  106.000  mm,	Z =   15.000 mm,
	W =-180.000 deg,	P =   0.000 deg,	R =    90.000 deg
};
P[5690]{
   GP1:
	UF : 1, UT : 5,		CONFIG : 'N U T, 0, 0, 0',
	X =  55.000  mm,	Y =  106.000  mm,	Z =   -1.000 mm,
	W =-180.000 deg,	P =   0.000 deg,	R =    90.000 deg
};
P[5691]{
   GP1:
	UF : 1, UT : 5,		CONFIG : 'N U T, 0, 0, 0',
	X =  55.000  mm,	Y =  106.000  mm,	Z =   15.000 mm,
	W =-180.000 deg,	P =   0.000 deg,	R =    90.000 deg
};
P[5692]{
   GP1:
	UF : 1, UT : 5,		CONFIG : 'N U T, 0, 0, 0',
	X =  73.000  mm,	Y =  106.000  mm,	Z =   15.000 mm,
	W =-180.000 deg,	P =   0.000 deg,	R =    90.000 deg
};
P[5693]{
   GP1:
	UF : 1, UT : 5,		CONFIG : 'N U T, 0, 0, 0',
	X =  73.000  mm,	Y =  106.000  mm,	Z =   -1.000 mm,
	W =-180.000 deg,	P =   0.000 deg,	R =    90.000 deg
};
P[5694]{
   GP1:
	UF : 1, UT : 5,		CONFIG : 'N U T, 0, 0, 0',
	X =  73.000  mm,	Y =  106.000  mm,	Z =   15.000 mm,
	W =-180.000 deg,	P =   0.000 deg,	R =    90.000 deg
};
P[5713]{
   GP1:
	UF : 1, UT : 5,		CONFIG : 'N U T, 0, 0, 0',
	X =  121.000  mm,	Y =  106.000  mm,	Z =   15.000 mm,
	W =-180.000 deg,	P =   0.000 deg,	R =    90.000 deg
};
P[5714]{
   GP1:
	UF : 1, UT : 5,		CONFIG : 'N U T, 0, 0, 0',
	X =  121.000  mm,	Y =  106.000  mm,	Z =   -1.000 mm,
	W =-180.000 deg,	P =   0.000 deg,	R =    90.000 deg
};
P[5715]{
   GP1:
	UF : 1, UT : 5,		CONFIG : 'N U T, 0, 0, 0',
	X =  121.000  mm,	Y =  106.000  mm,	Z =   15.000 mm,
	W =-180.000 deg,	P =   0.000 deg,	R =    90.000 deg
};
P[5716]{
   GP1:
	UF : 1, UT : 5,		CONFIG : 'N U T, 0, 0, 0',
	X =  124.000  mm,	Y =  106.000  mm,	Z =   15.000 mm,
	W =-180.000 deg,	P =   0.000 deg,	R =    90.000 deg
};
P[5717]{
   GP1:
	UF : 1, UT : 5,		CONFIG : 'N U T, 0, 0, 0',
	X =  124.000  mm,	Y =  106.000  mm,	Z =   -1.000 mm,
	W =-180.000 deg,	P =   0.000 deg,	R =    90.000 deg
};
P[5718]{
   GP1:
	UF : 1, UT : 5,		CONFIG : 'N U T, 0, 0, 0',
	X =  124.000  mm,	Y =  106.000  mm,	Z =   15.000 mm,
	W =-180.000 deg,	P =   0.000 deg,	R =    90.000 deg
};
P[5719]{
   GP1:
	UF : 1, UT : 5,		CONFIG : 'N U T, 0, 0, 0',
	X =  127.000  mm,	Y =  106.000  mm,	Z =   15.000 mm,
	W =-180.000 deg,	P =   0.000 deg,	R =    90.000 deg
};
P[5720]{
   GP1:
	UF : 1, UT : 5,		CONFIG : 'N U T, 0, 0, 0',
	X =  127.000  mm,	Y =  106.000  mm,	Z =   -1.000 mm,
	W =-180.000 deg,	P =   0.000 deg,	R =    90.000 deg
};
P[5721]{
   GP1:
	UF : 1, UT : 5,		CONFIG : 'N U T, 0, 0, 0',
	X =  127.000  mm,	Y =  106.000  mm,	Z =   15.000 mm,
	W =-180.000 deg,	P =   0.000 deg,	R =    90.000 deg
};
P[5722]{
   GP1:
	UF : 1, UT : 5,		CONFIG : 'N U T, 0, 0, 0',
	X =  130.000  mm,	Y =  106.000  mm,	Z =   15.000 mm,
	W =-180.000 deg,	P =   0.000 deg,	R =    90.000 deg
};
P[5723]{
   GP1:
	UF : 1, UT : 5,		CONFIG : 'N U T, 0, 0, 0',
	X =  130.000  mm,	Y =  106.000  mm,	Z =   -1.000 mm,
	W =-180.000 deg,	P =   0.000 deg,	R =    90.000 deg
};
P[5724]{
   GP1:
	UF : 1, UT : 5,		CONFIG : 'N U T, 0, 0, 0',
	X =  130.000  mm,	Y =  106.000  mm,	Z =   15.000 mm,
	W =-180.000 deg,	P =   0.000 deg,	R =    90.000 deg
};
P[5827]{
   GP1:
	UF : 1, UT : 5,		CONFIG : 'N U T, 0, 0, 0',
	X =  121.000  mm,	Y =  109.000  mm,	Z =   15.000 mm,
	W =-180.000 deg,	P =   0.000 deg,	R =    90.000 deg
};
P[5828]{
   GP1:
	UF : 1, UT : 5,		CONFIG : 'N U T, 0, 0, 0',
	X =  121.000  mm,	Y =  109.000  mm,	Z =   -1.000 mm,
	W =-180.000 deg,	P =   0.000 deg,	R =    90.000 deg
};
P[5829]{
   GP1:
	UF : 1, UT : 5,		CONFIG : 'N U T, 0, 0, 0',
	X =  121.000  mm,	Y =  109.000  mm,	Z =   15.000 mm,
	W =-180.000 deg,	P =   0.000 deg,	R =    90.000 deg
};
P[5830]{
   GP1:
	UF : 1, UT : 5,		CONFIG : 'N U T, 0, 0, 0',
	X =  124.000  mm,	Y =  109.000  mm,	Z =   15.000 mm,
	W =-180.000 deg,	P =   0.000 deg,	R =    90.000 deg
};
P[5831]{
   GP1:
	UF : 1, UT : 5,		CONFIG : 'N U T, 0, 0, 0',
	X =  124.000  mm,	Y =  109.000  mm,	Z =   -1.000 mm,
	W =-180.000 deg,	P =   0.000 deg,	R =    90.000 deg
};
P[5832]{
   GP1:
	UF : 1, UT : 5,		CONFIG : 'N U T, 0, 0, 0',
	X =  124.000  mm,	Y =  109.000  mm,	Z =   15.000 mm,
	W =-180.000 deg,	P =   0.000 deg,	R =    90.000 deg
};
P[5839]{
   GP1:
	UF : 1, UT : 5,		CONFIG : 'N U T, 0, 0, 0',
	X =  133.000  mm,	Y =  109.000  mm,	Z =   15.000 mm,
	W =-180.000 deg,	P =   0.000 deg,	R =    90.000 deg
};
P[5840]{
   GP1:
	UF : 1, UT : 5,		CONFIG : 'N U T, 0, 0, 0',
	X =  133.000  mm,	Y =  109.000  mm,	Z =   -1.000 mm,
	W =-180.000 deg,	P =   0.000 deg,	R =    90.000 deg
};
P[5841]{
   GP1:
	UF : 1, UT : 5,		CONFIG : 'N U T, 0, 0, 0',
	X =  133.000  mm,	Y =  109.000  mm,	Z =   15.000 mm,
	W =-180.000 deg,	P =   0.000 deg,	R =    90.000 deg
};
P[5926]{
   GP1:
	UF : 1, UT : 5,		CONFIG : 'N U T, 0, 0, 0',
	X =  121.000  mm,	Y =  112.000  mm,	Z =   15.000 mm,
	W =-180.000 deg,	P =   0.000 deg,	R =    90.000 deg
};
P[5927]{
   GP1:
	UF : 1, UT : 5,		CONFIG : 'N U T, 0, 0, 0',
	X =  121.000  mm,	Y =  112.000  mm,	Z =   -1.000 mm,
	W =-180.000 deg,	P =   0.000 deg,	R =    90.000 deg
};
P[5928]{
   GP1:
	UF : 1, UT : 5,		CONFIG : 'N U T, 0, 0, 0',
	X =  121.000  mm,	Y =  112.000  mm,	Z =   15.000 mm,
	W =-180.000 deg,	P =   0.000 deg,	R =    90.000 deg
};
P[6103]{
   GP1:
	UF : 1, UT : 5,		CONFIG : 'N U T, 0, 0, 0',
	X =  103.000  mm,	Y =  118.000  mm,	Z =   15.000 mm,
	W =-180.000 deg,	P =   0.000 deg,	R =    90.000 deg
};
P[6104]{
   GP1:
	UF : 1, UT : 5,		CONFIG : 'N U T, 0, 0, 0',
	X =  103.000  mm,	Y =  118.000  mm,	Z =   -1.000 mm,
	W =-180.000 deg,	P =   0.000 deg,	R =    90.000 deg
};
P[6105]{
   GP1:
	UF : 1, UT : 5,		CONFIG : 'N U T, 0, 0, 0',
	X =  103.000  mm,	Y =  118.000  mm,	Z =   15.000 mm,
	W =-180.000 deg,	P =   0.000 deg,	R =    90.000 deg
};
P[6208]{
   GP1:
	UF : 1, UT : 5,		CONFIG : 'N U T, 0, 0, 0',
	X =  103.000  mm,	Y =  121.000  mm,	Z =   15.000 mm,
	W =-180.000 deg,	P =   0.000 deg,	R =    90.000 deg
};
P[6209]{
   GP1:
	UF : 1, UT : 5,		CONFIG : 'N U T, 0, 0, 0',
	X =  103.000  mm,	Y =  121.000  mm,	Z =   -1.000 mm,
	W =-180.000 deg,	P =   0.000 deg,	R =    90.000 deg
};
P[6210]{
   GP1:
	UF : 1, UT : 5,		CONFIG : 'N U T, 0, 0, 0',
	X =  103.000  mm,	Y =  121.000  mm,	Z =   15.000 mm,
	W =-180.000 deg,	P =   0.000 deg,	R =    90.000 deg
};
P[6322]{
   GP1:
	UF : 1, UT : 5,		CONFIG : 'N U T, 0, 0, 0',
	X =  103.000  mm,	Y =  124.000  mm,	Z =   15.000 mm,
	W =-180.000 deg,	P =   0.000 deg,	R =    90.000 deg
};
P[6323]{
   GP1:
	UF : 1, UT : 5,		CONFIG : 'N U T, 0, 0, 0',
	X =  103.000  mm,	Y =  124.000  mm,	Z =   -1.000 mm,
	W =-180.000 deg,	P =   0.000 deg,	R =    90.000 deg
};
P[6324]{
   GP1:
	UF : 1, UT : 5,		CONFIG : 'N U T, 0, 0, 0',
	X =  103.000  mm,	Y =  124.000  mm,	Z =   15.000 mm,
	W =-180.000 deg,	P =   0.000 deg,	R =    90.000 deg
};
P[6430]{
   GP1:
	UF : 1, UT : 5,		CONFIG : 'N U T, 0, 0, 0',
	X =  67.000  mm,	Y =  127.000  mm,	Z =   15.000 mm,
	W =-180.000 deg,	P =   0.000 deg,	R =    90.000 deg
};
P[6431]{
   GP1:
	UF : 1, UT : 5,		CONFIG : 'N U T, 0, 0, 0',
	X =  67.000  mm,	Y =  127.000  mm,	Z =   -1.000 mm,
	W =-180.000 deg,	P =   0.000 deg,	R =    90.000 deg
};
P[6432]{
   GP1:
	UF : 1, UT : 5,		CONFIG : 'N U T, 0, 0, 0',
	X =  67.000  mm,	Y =  127.000  mm,	Z =   15.000 mm,
	W =-180.000 deg,	P =   0.000 deg,	R =    90.000 deg
};
P[6433]{
   GP1:
	UF : 1, UT : 5,		CONFIG : 'N U T, 0, 0, 0',
	X =  70.000  mm,	Y =  127.000  mm,	Z =   15.000 mm,
	W =-180.000 deg,	P =   0.000 deg,	R =    90.000 deg
};
P[6434]{
   GP1:
	UF : 1, UT : 5,		CONFIG : 'N U T, 0, 0, 0',
	X =  70.000  mm,	Y =  127.000  mm,	Z =   -1.000 mm,
	W =-180.000 deg,	P =   0.000 deg,	R =    90.000 deg
};
P[6435]{
   GP1:
	UF : 1, UT : 5,		CONFIG : 'N U T, 0, 0, 0',
	X =  70.000  mm,	Y =  127.000  mm,	Z =   15.000 mm,
	W =-180.000 deg,	P =   0.000 deg,	R =    90.000 deg
};
P[6436]{
   GP1:
	UF : 1, UT : 5,		CONFIG : 'N U T, 0, 0, 0',
	X =  73.000  mm,	Y =  127.000  mm,	Z =   15.000 mm,
	W =-180.000 deg,	P =   0.000 deg,	R =    90.000 deg
};
P[6437]{
   GP1:
	UF : 1, UT : 5,		CONFIG : 'N U T, 0, 0, 0',
	X =  73.000  mm,	Y =  127.000  mm,	Z =   -1.000 mm,
	W =-180.000 deg,	P =   0.000 deg,	R =    90.000 deg
};
P[6438]{
   GP1:
	UF : 1, UT : 5,		CONFIG : 'N U T, 0, 0, 0',
	X =  73.000  mm,	Y =  127.000  mm,	Z =   15.000 mm,
	W =-180.000 deg,	P =   0.000 deg,	R =    90.000 deg
};
P[6439]{
   GP1:
	UF : 1, UT : 5,		CONFIG : 'N U T, 0, 0, 0',
	X =  76.000  mm,	Y =  127.000  mm,	Z =   15.000 mm,
	W =-180.000 deg,	P =   0.000 deg,	R =    90.000 deg
};
P[6440]{
   GP1:
	UF : 1, UT : 5,		CONFIG : 'N U T, 0, 0, 0',
	X =  76.000  mm,	Y =  127.000  mm,	Z =   -1.000 mm,
	W =-180.000 deg,	P =   0.000 deg,	R =    90.000 deg
};
P[6441]{
   GP1:
	UF : 1, UT : 5,		CONFIG : 'N U T, 0, 0, 0',
	X =  76.000  mm,	Y =  127.000  mm,	Z =   15.000 mm,
	W =-180.000 deg,	P =   0.000 deg,	R =    90.000 deg
};
P[6442]{
   GP1:
	UF : 1, UT : 5,		CONFIG : 'N U T, 0, 0, 0',
	X =  79.000  mm,	Y =  127.000  mm,	Z =   15.000 mm,
	W =-180.000 deg,	P =   0.000 deg,	R =    90.000 deg
};
P[6443]{
   GP1:
	UF : 1, UT : 5,		CONFIG : 'N U T, 0, 0, 0',
	X =  79.000  mm,	Y =  127.000  mm,	Z =   -1.000 mm,
	W =-180.000 deg,	P =   0.000 deg,	R =    90.000 deg
};
P[6444]{
   GP1:
	UF : 1, UT : 5,		CONFIG : 'N U T, 0, 0, 0',
	X =  79.000  mm,	Y =  127.000  mm,	Z =   15.000 mm,
	W =-180.000 deg,	P =   0.000 deg,	R =    90.000 deg
};
P[6445]{
   GP1:
	UF : 1, UT : 5,		CONFIG : 'N U T, 0, 0, 0',
	X =  82.000  mm,	Y =  127.000  mm,	Z =   15.000 mm,
	W =-180.000 deg,	P =   0.000 deg,	R =    90.000 deg
};
P[6446]{
   GP1:
	UF : 1, UT : 5,		CONFIG : 'N U T, 0, 0, 0',
	X =  82.000  mm,	Y =  127.000  mm,	Z =   -1.000 mm,
	W =-180.000 deg,	P =   0.000 deg,	R =    90.000 deg
};
P[6447]{
   GP1:
	UF : 1, UT : 5,		CONFIG : 'N U T, 0, 0, 0',
	X =  82.000  mm,	Y =  127.000  mm,	Z =   15.000 mm,
	W =-180.000 deg,	P =   0.000 deg,	R =    90.000 deg
};
P[6448]{
   GP1:
	UF : 1, UT : 5,		CONFIG : 'N U T, 0, 0, 0',
	X =  103.000  mm,	Y =  127.000  mm,	Z =   15.000 mm,
	W =-180.000 deg,	P =   0.000 deg,	R =    90.000 deg
};
P[6449]{
   GP1:
	UF : 1, UT : 5,		CONFIG : 'N U T, 0, 0, 0',
	X =  103.000  mm,	Y =  127.000  mm,	Z =   -1.000 mm,
	W =-180.000 deg,	P =   0.000 deg,	R =    90.000 deg
};
P[6450]{
   GP1:
	UF : 1, UT : 5,		CONFIG : 'N U T, 0, 0, 0',
	X =  103.000  mm,	Y =  127.000  mm,	Z =   15.000 mm,
	W =-180.000 deg,	P =   0.000 deg,	R =    90.000 deg
};
P[6490]{
   GP1:
	UF : 1, UT : 5,		CONFIG : 'N U T, 0, 0, 0',
	X =  1.000  mm,	Y =  130.000  mm,	Z =   15.000 mm,
	W =-180.000 deg,	P =   0.000 deg,	R =    90.000 deg
};
P[6491]{
   GP1:
	UF : 1, UT : 5,		CONFIG : 'N U T, 0, 0, 0',
	X =  1.000  mm,	Y =  130.000  mm,	Z =   -1.000 mm,
	W =-180.000 deg,	P =   0.000 deg,	R =    90.000 deg
};
P[6492]{
   GP1:
	UF : 1, UT : 5,		CONFIG : 'N U T, 0, 0, 0',
	X =  1.000  mm,	Y =  130.000  mm,	Z =   15.000 mm,
	W =-180.000 deg,	P =   0.000 deg,	R =    90.000 deg
};
P[6493]{
   GP1:
	UF : 1, UT : 5,		CONFIG : 'N U T, 0, 0, 0',
	X =  4.000  mm,	Y =  130.000  mm,	Z =   15.000 mm,
	W =-180.000 deg,	P =   0.000 deg,	R =    90.000 deg
};
P[6494]{
   GP1:
	UF : 1, UT : 5,		CONFIG : 'N U T, 0, 0, 0',
	X =  4.000  mm,	Y =  130.000  mm,	Z =   -1.000 mm,
	W =-180.000 deg,	P =   0.000 deg,	R =    90.000 deg
};
P[6495]{
   GP1:
	UF : 1, UT : 5,		CONFIG : 'N U T, 0, 0, 0',
	X =  4.000  mm,	Y =  130.000  mm,	Z =   15.000 mm,
	W =-180.000 deg,	P =   0.000 deg,	R =    90.000 deg
};
P[6499]{
   GP1:
	UF : 1, UT : 5,		CONFIG : 'N U T, 0, 0, 0',
	X =  10.000  mm,	Y =  130.000  mm,	Z =   15.000 mm,
	W =-180.000 deg,	P =   0.000 deg,	R =    90.000 deg
};
P[6500]{
   GP1:
	UF : 1, UT : 5,		CONFIG : 'N U T, 0, 0, 0',
	X =  10.000  mm,	Y =  130.000  mm,	Z =   -1.000 mm,
	W =-180.000 deg,	P =   0.000 deg,	R =    90.000 deg
};
P[6501]{
   GP1:
	UF : 1, UT : 5,		CONFIG : 'N U T, 0, 0, 0',
	X =  10.000  mm,	Y =  130.000  mm,	Z =   15.000 mm,
	W =-180.000 deg,	P =   0.000 deg,	R =    90.000 deg
};
P[6502]{
   GP1:
	UF : 1, UT : 5,		CONFIG : 'N U T, 0, 0, 0',
	X =  13.000  mm,	Y =  130.000  mm,	Z =   15.000 mm,
	W =-180.000 deg,	P =   0.000 deg,	R =    90.000 deg
};
P[6503]{
   GP1:
	UF : 1, UT : 5,		CONFIG : 'N U T, 0, 0, 0',
	X =  13.000  mm,	Y =  130.000  mm,	Z =   -1.000 mm,
	W =-180.000 deg,	P =   0.000 deg,	R =    90.000 deg
};
P[6504]{
   GP1:
	UF : 1, UT : 5,		CONFIG : 'N U T, 0, 0, 0',
	X =  13.000  mm,	Y =  130.000  mm,	Z =   15.000 mm,
	W =-180.000 deg,	P =   0.000 deg,	R =    90.000 deg
};
P[6553]{
   GP1:
	UF : 1, UT : 5,		CONFIG : 'N U T, 0, 0, 0',
	X =  103.000  mm,	Y =  130.000  mm,	Z =   15.000 mm,
	W =-180.000 deg,	P =   0.000 deg,	R =    90.000 deg
};
P[6554]{
   GP1:
	UF : 1, UT : 5,		CONFIG : 'N U T, 0, 0, 0',
	X =  103.000  mm,	Y =  130.000  mm,	Z =   -1.000 mm,
	W =-180.000 deg,	P =   0.000 deg,	R =    90.000 deg
};
P[6555]{
   GP1:
	UF : 1, UT : 5,		CONFIG : 'N U T, 0, 0, 0',
	X =  103.000  mm,	Y =  130.000  mm,	Z =   15.000 mm,
	W =-180.000 deg,	P =   0.000 deg,	R =    90.000 deg
};
P[6598]{
   GP1:
	UF : 1, UT : 5,		CONFIG : 'N U T, 0, 0, 0',
	X =  154.000  mm,	Y =  130.000  mm,	Z =   15.000 mm,
	W =-180.000 deg,	P =   0.000 deg,	R =    90.000 deg
};
P[6599]{
   GP1:
	UF : 1, UT : 5,		CONFIG : 'N U T, 0, 0, 0',
	X =  154.000  mm,	Y =  130.000  mm,	Z =   -1.000 mm,
	W =-180.000 deg,	P =   0.000 deg,	R =    90.000 deg
};
P[6600]{
   GP1:
	UF : 1, UT : 5,		CONFIG : 'N U T, 0, 0, 0',
	X =  154.000  mm,	Y =  130.000  mm,	Z =   15.000 mm,
	W =-180.000 deg,	P =   0.000 deg,	R =    90.000 deg
};
P[6610]{
   GP1:
	UF : 1, UT : 5,		CONFIG : 'N U T, 0, 0, 0',
	X =  166.000  mm,	Y =  130.000  mm,	Z =   15.000 mm,
	W =-180.000 deg,	P =   0.000 deg,	R =    90.000 deg
};
P[6611]{
   GP1:
	UF : 1, UT : 5,		CONFIG : 'N U T, 0, 0, 0',
	X =  166.000  mm,	Y =  130.000  mm,	Z =   -1.000 mm,
	W =-180.000 deg,	P =   0.000 deg,	R =    90.000 deg
};
P[6612]{
   GP1:
	UF : 1, UT : 5,		CONFIG : 'N U T, 0, 0, 0',
	X =  166.000  mm,	Y =  130.000  mm,	Z =   15.000 mm,
	W =-180.000 deg,	P =   0.000 deg,	R =    90.000 deg
};
P[6613]{
   GP1:
	UF : 1, UT : 5,		CONFIG : 'N U T, 0, 0, 0',
	X =  169.000  mm,	Y =  130.000  mm,	Z =   15.000 mm,
	W =-180.000 deg,	P =   0.000 deg,	R =    90.000 deg
};
P[6614]{
   GP1:
	UF : 1, UT : 5,		CONFIG : 'N U T, 0, 0, 0',
	X =  169.000  mm,	Y =  130.000  mm,	Z =   -1.000 mm,
	W =-180.000 deg,	P =   0.000 deg,	R =    90.000 deg
};
P[6615]{
   GP1:
	UF : 1, UT : 5,		CONFIG : 'N U T, 0, 0, 0',
	X =  169.000  mm,	Y =  130.000  mm,	Z =   15.000 mm,
	W =-180.000 deg,	P =   0.000 deg,	R =    90.000 deg
};
P[6616]{
   GP1:
	UF : 1, UT : 5,		CONFIG : 'N U T, 0, 0, 0',
	X =  172.000  mm,	Y =  130.000  mm,	Z =   15.000 mm,
	W =-180.000 deg,	P =   0.000 deg,	R =    90.000 deg
};
P[6617]{
   GP1:
	UF : 1, UT : 5,		CONFIG : 'N U T, 0, 0, 0',
	X =  172.000  mm,	Y =  130.000  mm,	Z =   -1.000 mm,
	W =-180.000 deg,	P =   0.000 deg,	R =    90.000 deg
};
P[6618]{
   GP1:
	UF : 1, UT : 5,		CONFIG : 'N U T, 0, 0, 0',
	X =  172.000  mm,	Y =  130.000  mm,	Z =   15.000 mm,
	W =-180.000 deg,	P =   0.000 deg,	R =    90.000 deg
};
P[6619]{
   GP1:
	UF : 1, UT : 5,		CONFIG : 'N U T, 0, 0, 0',
	X =  175.000  mm,	Y =  130.000  mm,	Z =   15.000 mm,
	W =-180.000 deg,	P =   0.000 deg,	R =    90.000 deg
};
P[6620]{
   GP1:
	UF : 1, UT : 5,		CONFIG : 'N U T, 0, 0, 0',
	X =  175.000  mm,	Y =  130.000  mm,	Z =   -1.000 mm,
	W =-180.000 deg,	P =   0.000 deg,	R =    90.000 deg
};
P[6621]{
   GP1:
	UF : 1, UT : 5,		CONFIG : 'N U T, 0, 0, 0',
	X =  175.000  mm,	Y =  130.000  mm,	Z =   15.000 mm,
	W =-180.000 deg,	P =   0.000 deg,	R =    90.000 deg
};
P[6676]{
   GP1:
	UF : 1, UT : 5,		CONFIG : 'N U T, 0, 0, 0',
	X =  106.000  mm,	Y =  133.000  mm,	Z =   15.000 mm,
	W =-180.000 deg,	P =   0.000 deg,	R =    90.000 deg
};
P[6677]{
   GP1:
	UF : 1, UT : 5,		CONFIG : 'N U T, 0, 0, 0',
	X =  106.000  mm,	Y =  133.000  mm,	Z =   -1.000 mm,
	W =-180.000 deg,	P =   0.000 deg,	R =    90.000 deg
};
P[6678]{
   GP1:
	UF : 1, UT : 5,		CONFIG : 'N U T, 0, 0, 0',
	X =  106.000  mm,	Y =  133.000  mm,	Z =   15.000 mm,
	W =-180.000 deg,	P =   0.000 deg,	R =    90.000 deg
};
P[6727]{
   GP1:
	UF : 1, UT : 5,		CONFIG : 'N U T, 0, 0, 0',
	X =  157.000  mm,	Y =  133.000  mm,	Z =   15.000 mm,
	W =-180.000 deg,	P =   0.000 deg,	R =    90.000 deg
};
P[6728]{
   GP1:
	UF : 1, UT : 5,		CONFIG : 'N U T, 0, 0, 0',
	X =  157.000  mm,	Y =  133.000  mm,	Z =   -1.000 mm,
	W =-180.000 deg,	P =   0.000 deg,	R =    90.000 deg
};
P[6729]{
   GP1:
	UF : 1, UT : 5,		CONFIG : 'N U T, 0, 0, 0',
	X =  157.000  mm,	Y =  133.000  mm,	Z =   15.000 mm,
	W =-180.000 deg,	P =   0.000 deg,	R =    90.000 deg
};
P[6826]{
   GP1:
	UF : 1, UT : 5,		CONFIG : 'N U T, 0, 0, 0',
	X =  157.000  mm,	Y =  136.000  mm,	Z =   15.000 mm,
	W =-180.000 deg,	P =   0.000 deg,	R =    90.000 deg
};
P[6827]{
   GP1:
	UF : 1, UT : 5,		CONFIG : 'N U T, 0, 0, 0',
	X =  157.000  mm,	Y =  136.000  mm,	Z =   -1.000 mm,
